    movel([0.504361, -1.310843, -2.623001, -0.778545, 1.570796, 2.075158],accel_mss,speed_ms,0,blend_radius_m)
    movel([0.505882, -1.309678, -2.623708, -0.779003, 1.570796, 2.076678],accel_mss,speed_ms,0,blend_radius_m)
    movel([0.507291, -1.308414, -2.624472, -0.779502, 1.570796, 2.078088],accel_mss,speed_ms,0,blend_radius_m)
    movel([0.508613, -1.307071, -2.625283, -0.780035, 1.570796, 2.079409],accel_mss,speed_ms,0,blend_radius_m)
    movel([0.509871, -1.305667, -2.626128, -0.780594, 1.570796, 2.080667],accel_mss,speed_ms,0,blend_radius_m)
    movel([0.514730, -1.299885, -2.629580, -0.782925, 1.570796, 2.085526],accel_mss,speed_ms,0,blend_radius_m)
    movel([0.516568, -1.297775, -2.630828, -0.783786, 1.570796, 2.087364],accel_mss,speed_ms,0,blend_radius_m)
    movel([0.518895, -1.295391, -2.632232, -0.784766, 1.570796, 2.089692],accel_mss,speed_ms,0,blend_radius_m)
    movel([0.520143, -1.294383, -2.632824, -0.785183, 1.570796, 2.090940],accel_mss,speed_ms,0,blend_radius_m)
    movel([0.521391, -1.293655, -2.633250, -0.785484, 1.570796, 2.092187],accel_mss,speed_ms,0,blend_radius_m)
    movel([0.522003, -1.293434, -2.633379, -0.785576, 1.570796, 2.092800],accel_mss,speed_ms,0,blend_radius_m)
    movel([0.523177, -1.293343, -2.633433, -0.785614, 1.570796, 2.093973],accel_mss,speed_ms,0,blend_radius_m)
    movel([0.523727, -1.293507, -2.633336, -0.785546, 1.570796, 2.094523],accel_mss,speed_ms,0,blend_radius_m)
    movel([0.524119, -1.293909, -2.633101, -0.785379, 1.570796, 2.094915],accel_mss,speed_ms,0,blend_radius_m)
    movel([0.524203, -1.294537, -2.632733, -0.785119, 1.570796, 2.095000],accel_mss,speed_ms,0,blend_radius_m)
    movel([0.523804, -1.296075, -2.631830, -0.784484, 1.570796, 2.094600],accel_mss,speed_ms,0,blend_radius_m)
    movel([0.522876, -1.298205, -2.630574, -0.783610, 1.570796, 2.093672],accel_mss,speed_ms,0,blend_radius_m)
    movel([0.521782, -1.300323, -2.629319, -0.782746, 1.570796, 2.092578],accel_mss,speed_ms,0,blend_radius_m)
    movel([0.523955, -1.298870, -2.630181, -0.783338, 1.570796, 2.094752],accel_mss,speed_ms,0,blend_radius_m)
    movel([0.526201, -1.297582, -2.630942, -0.783865, 1.570796, 2.096997],accel_mss,speed_ms,0,blend_radius_m)
    movel([0.528485, -1.296466, -2.631600, -0.784323, 1.570796, 2.099281],accel_mss,speed_ms,0,blend_radius_m)
    movel([0.530768, -1.295526, -2.632153, -0.784710, 1.570796, 2.101564],accel_mss,speed_ms,0,blend_radius_m)
    movel([0.535321, -1.293655, -2.633250, -0.785484, 1.570796, 2.106117],accel_mss,speed_ms,0,blend_radius_m)
    movel([0.536592, -1.293226, -2.633501, -0.785662, 1.570796, 2.107388],accel_mss,speed_ms,0,blend_radius_m)
    movel([0.537753, -1.292944, -2.633665, -0.785779, 1.570796, 2.108550],accel_mss,speed_ms,0,blend_radius_m)
    movel([0.538730, -1.292873, -2.633707, -0.785809, 1.570796, 2.109526],accel_mss,speed_ms,0,blend_radius_m)
    movel([0.539439, -1.293071, -2.633591, -0.785727, 1.570796, 2.110235],accel_mss,speed_ms,0,blend_radius_m)
    movel([0.539796, -1.293629, -2.633265, -0.785495, 1.570796, 2.110592],accel_mss,speed_ms,0,blend_radius_m)
    movel([0.539763, -1.294477, -2.632768, -0.785143, 1.570796, 2.110560],accel_mss,speed_ms,0,blend_radius_m)
    movel([0.539417, -1.295518, -2.632157, -0.784713, 1.570796, 2.110214],accel_mss,speed_ms,0,blend_radius_m)
    movel([0.538829, -1.296650, -2.631491, -0.784247, 1.570796, 2.109626],accel_mss,speed_ms,0,blend_radius_m)
    movel([0.538074, -1.297775, -2.630828, -0.783786, 1.570796, 2.108870],accel_mss,speed_ms,0,blend_radius_m)
    movel([0.537226, -1.298794, -2.630226, -0.783369, 1.570796, 2.108023],accel_mss,speed_ms,0,blend_radius_m)
    movel([0.536357, -1.299608, -2.629743, -0.783037, 1.570796, 2.107154],accel_mss,speed_ms,0,blend_radius_m)
    movel([0.535539, -1.300121, -2.629439, -0.782829, 1.570796, 2.106335],accel_mss,speed_ms,0,blend_radius_m)
    movel([0.539564, -1.298618, -2.630330, -0.783441, 1.570796, 2.110360],accel_mss,speed_ms,0,blend_radius_m)
    movel([0.541559, -1.298052, -2.630664, -0.783672, 1.570796, 2.112356],accel_mss,speed_ms,0,blend_radius_m)
    movel([0.543523, -1.297629, -2.630915, -0.783846, 1.570796, 2.114320],accel_mss,speed_ms,0,blend_radius_m)
    movel([0.545439, -1.297358, -2.631074, -0.783957, 1.570796, 2.116236],accel_mss,speed_ms,0,blend_radius_m)
    movel([0.547294, -1.297255, -2.631135, -0.783999, 1.570796, 2.118090],accel_mss,speed_ms,0,blend_radius_m)
    movel([0.549070, -1.297333, -2.631089, -0.783967, 1.570796, 2.119867],accel_mss,speed_ms,0,blend_radius_m)
    movel([0.550755, -1.297601, -2.630931, -0.783857, 1.570796, 2.121552],accel_mss,speed_ms,0,blend_radius_m)
    movel([0.551714, -1.298079, -2.630649, -0.783661, 1.570796, 2.122511],accel_mss,speed_ms,0,blend_radius_m)
    movel([0.552495, -1.298983, -2.630114, -0.783292, 1.570796, 2.123291],accel_mss,speed_ms,0,blend_radius_m)
    movel([0.552726, -1.299550, -2.629778, -0.783061, 1.570796, 2.123522],accel_mss,speed_ms,0,blend_radius_m)
    movel([0.552803, -1.300169, -2.629411, -0.782809, 1.570796, 2.123599],accel_mss,speed_ms,0,blend_radius_m)
    movel([0.552691, -1.300824, -2.629021, -0.782543, 1.570796, 2.123487],accel_mss,speed_ms,0,blend_radius_m)
    movel([0.552350, -1.301497, -2.628621, -0.782270, 1.570796, 2.123146],accel_mss,speed_ms,0,blend_radius_m)
    movel([0.551814, -1.302079, -2.628275, -0.782035, 1.570796, 2.122610],accel_mss,speed_ms,0,blend_radius_m)
    movel([0.551157, -1.302554, -2.627992, -0.781844, 1.570796, 2.121954],accel_mss,speed_ms,0,blend_radius_m)
    movel([0.549592, -1.303332, -2.627527, -0.781530, 1.570796, 2.120389],accel_mss,speed_ms,0,blend_radius_m)
    movel([0.548029, -1.303757, -2.627273, -0.781359, 1.570796, 2.118825],accel_mss,speed_ms,0,blend_radius_m)
    movel([0.546506, -1.303910, -2.627181, -0.781298, 1.570796, 2.117302],accel_mss,speed_ms,0,blend_radius_m)
    movel([0.545064, -1.303868, -2.627206, -0.781315, 1.570796, 2.115860],accel_mss,speed_ms,0,blend_radius_m)
    movel([0.546236, -1.305031, -2.626509, -0.780848, 1.570796, 2.117032],accel_mss,speed_ms,0,blend_radius_m)
    movel([0.547593, -1.306014, -2.625919, -0.780456, 1.570796, 2.118389],accel_mss,speed_ms,0,blend_radius_m)
    movel([0.549117, -1.306810, -2.625440, -0.780139, 1.570796, 2.119913],accel_mss,speed_ms,0,blend_radius_m)
    movel([0.550792, -1.307414, -2.625076, -0.779899, 1.570796, 2.121588],accel_mss,speed_ms,0,blend_radius_m)
    movel([0.552231, -1.307696, -2.624906, -0.779787, 1.570796, 2.123027],accel_mss,speed_ms,0,blend_radius_m)
    movel([0.555218, -1.307960, -2.624746, -0.779682, 1.570796, 2.126015],accel_mss,speed_ms,0,blend_radius_m)
    movel([0.556664, -1.308230, -2.624584, -0.779575, 1.570796, 2.127460],accel_mss,speed_ms,0,blend_radius_m)
    movel([0.558212, -1.308690, -2.624306, -0.779393, 1.570796, 2.129009],accel_mss,speed_ms,0,blend_radius_m)
    movel([0.560696, -1.309649, -2.623725, -0.779015, 1.570796, 2.131492],accel_mss,speed_ms,0,blend_radius_m)
    movel([0.561790, -1.310255, -2.623358, -0.778776, 1.570796, 2.132586],accel_mss,speed_ms,0,blend_radius_m)
    movel([0.562521, -1.310911, -2.622960, -0.778519, 1.570796, 2.133318],accel_mss,speed_ms,0,blend_radius_m)
    movel([0.562691, -1.311249, -2.622754, -0.778386, 1.570796, 2.133487],accel_mss,speed_ms,0,blend_radius_m)
    movel([0.562694, -1.311591, -2.622546, -0.778252, 1.570796, 2.133490],accel_mss,speed_ms,0,blend_radius_m)
    movel([0.562510, -1.311931, -2.622339, -0.778119, 1.570796, 2.133307],accel_mss,speed_ms,0,blend_radius_m)
    movel([0.562113, -1.312265, -2.622135, -0.777989, 1.570796, 2.132910],accel_mss,speed_ms,0,blend_radius_m)
    movel([0.561025, -1.312830, -2.621791, -0.777768, 1.570796, 2.131822],accel_mss,speed_ms,0,blend_radius_m)
    movel([0.559815, -1.313224, -2.621550, -0.777614, 1.570796, 2.130611],accel_mss,speed_ms,0,blend_radius_m)
    movel([0.558524, -1.313482, -2.621393, -0.777514, 1.570796, 2.129320],accel_mss,speed_ms,0,blend_radius_m)
    movel([0.557205, -1.313629, -2.621303, -0.777457, 1.570796, 2.128001],accel_mss,speed_ms,0,blend_radius_m)
    movel([0.554665, -1.313702, -2.621258, -0.777429, 1.570796, 2.125461],accel_mss,speed_ms,0,blend_radius_m)
    movel([0.552577, -1.313666, -2.621280, -0.777443, 1.570796, 2.123374],accel_mss,speed_ms,0,blend_radius_m)
    movel([0.553095, -1.314568, -2.620728, -0.777093, 1.570796, 2.123892],accel_mss,speed_ms,0,blend_radius_m)
    movel([0.553726, -1.315378, -2.620232, -0.776779, 1.570796, 2.124522],accel_mss,speed_ms,0,blend_radius_m)
    movel([0.555262, -1.316761, -2.619382, -0.776246, 1.570796, 2.126058],accel_mss,speed_ms,0,blend_radius_m)
    movel([0.557070, -1.317890, -2.618687, -0.775813, 1.570796, 2.127867],accel_mss,speed_ms,0,blend_radius_m)
    movel([0.559036, -1.318840, -2.618100, -0.775449, 1.570796, 2.129832],accel_mss,speed_ms,0,blend_radius_m)
    movel([0.560750, -1.319486, -2.617700, -0.775203, 1.570796, 2.131546],accel_mss,speed_ms,0,blend_radius_m)
    movel([0.566077, -1.321158, -2.616663, -0.774568, 1.570796, 2.136873],accel_mss,speed_ms,0,blend_radius_m)
    movel([0.566925, -1.321690, -2.616333, -0.774366, 1.570796, 2.137721],accel_mss,speed_ms,0,blend_radius_m)
    movel([0.567404, -1.322414, -2.615882, -0.774093, 1.570796, 2.138201],accel_mss,speed_ms,0,blend_radius_m)
    movel([0.567376, -1.322780, -2.615654, -0.773955, 1.570796, 2.138172],accel_mss,speed_ms,0,blend_radius_m)
    movel([0.567099, -1.323110, -2.615448, -0.773831, 1.570796, 2.137895],accel_mss,speed_ms,0,blend_radius_m)
    movel([0.566520, -1.323378, -2.615281, -0.773730, 1.570796, 2.137317],accel_mss,speed_ms,0,blend_radius_m)
    movel([0.565588, -1.323554, -2.615171, -0.773664, 1.570796, 2.136384],accel_mss,speed_ms,0,blend_radius_m)
    movel([0.564160, -1.323615, -2.615133, -0.773641, 1.570796, 2.134956],accel_mss,speed_ms,0,blend_radius_m)
    movel([0.562620, -1.323495, -2.615208, -0.773686, 1.570796, 2.133416],accel_mss,speed_ms,0,blend_radius_m)
    movel([0.561231, -1.323153, -2.615421, -0.773815, 1.570796, 2.132027],accel_mss,speed_ms,0,blend_radius_m)
    movel([0.560674, -1.322887, -2.615587, -0.773915, 1.570796, 2.131470],accel_mss,speed_ms,0,blend_radius_m)
    movel([0.560257, -1.322548, -2.615798, -0.774042, 1.570796, 2.131053],accel_mss,speed_ms,0,blend_radius_m)
    movel([0.561241, -1.324942, -2.614303, -0.773144, 1.570796, 2.132038],accel_mss,speed_ms,0,blend_radius_m)
    movel([0.562524, -1.327120, -2.612935, -0.772333, 1.570796, 2.133321],accel_mss,speed_ms,0,blend_radius_m)
    movel([0.564045, -1.329119, -2.611675, -0.771595, 1.570796, 2.134841],accel_mss,speed_ms,0,blend_radius_m)
    movel([0.565745, -1.330982, -2.610496, -0.770912, 1.570796, 2.136541],accel_mss,speed_ms,0,blend_radius_m)
    movel([0.569451, -1.334431, -2.608299, -0.769659, 1.570796, 2.140247],accel_mss,speed_ms,0,blend_radius_m)
    movel([0.573175, -1.337754, -2.606167, -0.768468, 1.570796, 2.143972],accel_mss,speed_ms,0,blend_radius_m)
    movel([0.573691, -1.338478, -2.605701, -0.768210, 1.570796, 2.144487],accel_mss,speed_ms,0,blend_radius_m)
    movel([0.573735, -1.338932, -2.605408, -0.768049, 1.570796, 2.144531],accel_mss,speed_ms,0,blend_radius_m)
    movel([0.573528, -1.339439, -2.605080, -0.767869, 1.570796, 2.144324],accel_mss,speed_ms,0,blend_radius_m)
    movel([0.573099, -1.339888, -2.604790, -0.767711, 1.570796, 2.143896],accel_mss,speed_ms,0,blend_radius_m)
    movel([0.571722, -1.340678, -2.604279, -0.767432, 1.570796, 2.142518],accel_mss,speed_ms,0,blend_radius_m)
    movel([0.570874, -1.341000, -2.604070, -0.767318, 1.570796, 2.141670],accel_mss,speed_ms,0,blend_radius_m)
    movel([0.569183, -1.341339, -2.603851, -0.767199, 1.570796, 2.139979],accel_mss,speed_ms,0,blend_radius_m)
    movel([0.567539, -1.341325, -2.603860, -0.767204, 1.570796, 2.138335],accel_mss,speed_ms,0,blend_radius_m)
    movel([0.565973, -1.341026, -2.604053, -0.767309, 1.570796, 2.136769],accel_mss,speed_ms,0,blend_radius_m)
    movel([0.564526, -1.340506, -2.604390, -0.767492, 1.570796, 2.135323],accel_mss,speed_ms,0,blend_radius_m)
    movel([0.563234, -1.339833, -2.604826, -0.767730, 1.570796, 2.134030],accel_mss,speed_ms,0,blend_radius_m)
    movel([0.562135, -1.339068, -2.605320, -0.768001, 1.570796, 2.132931],accel_mss,speed_ms,0,blend_radius_m)
    movel([0.561270, -1.338276, -2.605831, -0.768282, 1.570796, 2.132067],accel_mss,speed_ms,0,blend_radius_m)
    movel([0.561003, -1.338714, -2.605548, -0.768126, 1.570796, 2.131799],accel_mss,speed_ms,0,blend_radius_m)
    movel([0.560974, -1.339164, -2.605258, -0.767967, 1.570796, 2.131770],accel_mss,speed_ms,0,blend_radius_m)
    movel([0.561152, -1.340097, -2.604655, -0.767637, 1.570796, 2.131948],accel_mss,speed_ms,0,blend_radius_m)
    movel([0.561472, -1.340950, -2.604103, -0.767336, 1.570796, 2.132269],accel_mss,speed_ms,0,blend_radius_m)
    movel([0.562363, -1.342502, -2.603095, -0.766792, 1.570796, 2.133160],accel_mss,speed_ms,0,blend_radius_m)
    movel([0.564091, -1.345024, -2.601451, -0.765914, 1.570796, 2.134887],accel_mss,speed_ms,0,blend_radius_m)
    movel([0.565937, -1.347426, -2.599877, -0.765086, 1.570796, 2.136734],accel_mss,speed_ms,0,blend_radius_m)
    movel([0.569942, -1.351936, -2.596899, -0.763554, 1.570796, 2.140738],accel_mss,speed_ms,0,blend_radius_m)
    movel([0.571032, -1.353216, -2.596049, -0.763124, 1.570796, 2.141829],accel_mss,speed_ms,0,blend_radius_m)
    movel([0.571656, -1.354143, -2.595432, -0.762814, 1.570796, 2.142452],accel_mss,speed_ms,0,blend_radius_m)
    movel([0.572170, -1.355176, -2.594743, -0.762470, 1.570796, 2.142967],accel_mss,speed_ms,0,blend_radius_m)
    movel([0.572449, -1.356251, -2.594024, -0.762114, 1.570796, 2.143245],accel_mss,speed_ms,0,blend_radius_m)
    movel([0.572374, -1.357299, -2.593321, -0.761768, 1.570796, 2.143170],accel_mss,speed_ms,0,blend_radius_m)
    movel([0.572168, -1.357794, -2.592990, -0.761606, 1.570796, 2.142964],accel_mss,speed_ms,0,blend_radius_m)
    movel([0.571829, -1.358259, -2.592677, -0.761453, 1.570796, 2.142626],accel_mss,speed_ms,0,blend_radius_m)
    movel([0.571338, -1.358686, -2.592390, -0.761313, 1.570796, 2.142135],accel_mss,speed_ms,0,blend_radius_m)
    movel([0.570686, -1.359068, -2.592133, -0.761188, 1.570796, 2.141483],accel_mss,speed_ms,0,blend_radius_m)
    movel([0.569974, -1.359179, -2.592058, -0.761152, 1.570796, 2.140771],accel_mss,speed_ms,0,blend_radius_m)
    movel([0.569174, -1.359018, -2.592167, -0.761205, 1.570796, 2.139971],accel_mss,speed_ms,0,blend_radius_m)
    movel([0.565202, -1.357551, -2.593152, -0.761685, 1.570796, 2.135998],accel_mss,speed_ms,0,blend_radius_m)
    movel([0.563995, -1.356820, -2.593642, -0.761926, 1.570796, 2.134792],accel_mss,speed_ms,0,blend_radius_m)
    movel([0.563549, -1.356378, -2.593939, -0.762072, 1.570796, 2.134345],accel_mss,speed_ms,0,blend_radius_m)
    movel([0.563259, -1.355871, -2.594278, -0.762240, 1.570796, 2.134055],accel_mss,speed_ms,0,blend_radius_m)
    movel([0.563894, -1.359000, -2.592178, -0.761210, 1.570796, 2.134690],accel_mss,speed_ms,0,blend_radius_m)
    movel([0.564930, -1.361895, -2.590224, -0.760271, 1.570796, 2.135727],accel_mss,speed_ms,0,blend_radius_m)
    movel([0.566288, -1.364581, -2.588399, -0.759409, 1.570796, 2.137084],accel_mss,speed_ms,0,blend_radius_m)
    movel([0.567890, -1.367082, -2.586691, -0.758616, 1.570796, 2.138687],accel_mss,speed_ms,0,blend_radius_m)
    movel([0.569508, -1.368812, -2.585505, -0.758073, 1.570796, 2.140304],accel_mss,speed_ms,0,blend_radius_m)
    movel([0.571786, -1.371355, -2.583753, -0.757281, 1.570796, 2.142582],accel_mss,speed_ms,0,blend_radius_m)
    movel([0.572698, -1.372726, -2.582804, -0.756859, 1.570796, 2.143494],accel_mss,speed_ms,0,blend_radius_m)
    movel([0.573213, -1.374054, -2.581883, -0.756452, 1.570796, 2.144009],accel_mss,speed_ms,0,blend_radius_m)
    movel([0.573263, -1.374675, -2.581452, -0.756263, 1.570796, 2.144060],accel_mss,speed_ms,0,blend_radius_m)
    movel([0.573144, -1.375252, -2.581050, -0.756087, 1.570796, 2.143941],accel_mss,speed_ms,0,blend_radius_m)
    movel([0.572832, -1.375778, -2.580683, -0.755928, 1.570796, 2.143628],accel_mss,speed_ms,0,blend_radius_m)
    movel([0.572309, -1.376242, -2.580360, -0.755787, 1.570796, 2.143105],accel_mss,speed_ms,0,blend_radius_m)
    movel([0.571702, -1.376584, -2.580121, -0.755684, 1.570796, 2.142498],accel_mss,speed_ms,0,blend_radius_m)
    movel([0.571079, -1.376828, -2.579951, -0.755610, 1.570796, 2.141875],accel_mss,speed_ms,0,blend_radius_m)
    movel([0.569831, -1.377119, -2.579747, -0.755523, 1.570796, 2.140627],accel_mss,speed_ms,0,blend_radius_m)
    movel([0.568531, -1.377283, -2.579632, -0.755473, 1.570796, 2.139327],accel_mss,speed_ms,0,blend_radius_m)
    movel([0.566060, -1.377286, -2.579631, -0.755473, 1.570796, 2.136857],accel_mss,speed_ms,0,blend_radius_m)
    movel([0.564904, -1.377127, -2.579742, -0.755520, 1.570796, 2.135700],accel_mss,speed_ms,0,blend_radius_m)
    movel([0.566200, -1.378941, -2.578471, -0.754977, 1.570796, 2.136997],accel_mss,speed_ms,0,blend_radius_m)
    movel([0.567641, -1.380619, -2.577292, -0.754478, 1.570796, 2.138437],accel_mss,speed_ms,0,blend_radius_m)
    movel([0.569208, -1.382177, -2.576193, -0.754019, 1.570796, 2.140004],accel_mss,speed_ms,0,blend_radius_m)
    movel([0.570887, -1.383627, -2.575167, -0.753594, 1.570796, 2.141683],accel_mss,speed_ms,0,blend_radius_m)
    movel([0.574515, -1.386268, -2.573291, -0.752829, 1.570796, 2.145311],accel_mss,speed_ms,0,blend_radius_m)
    movel([0.578407, -1.388652, -2.571589, -0.752148, 1.570796, 2.149203],accel_mss,speed_ms,0,blend_radius_m)
    movel([0.579346, -1.389428, -2.571034, -0.751928, 1.570796, 2.150143],accel_mss,speed_ms,0,blend_radius_m)
    movel([0.579550, -1.389960, -2.570652, -0.751777, 1.570796, 2.150347],accel_mss,speed_ms,0,blend_radius_m)
    movel([0.579414, -1.390611, -2.570185, -0.751594, 1.570796, 2.150210],accel_mss,speed_ms,0,blend_radius_m)
    movel([0.579137, -1.391041, -2.569875, -0.751473, 1.570796, 2.149933],accel_mss,speed_ms,0,blend_radius_m)
    movel([0.578763, -1.391416, -2.569605, -0.751367, 1.570796, 2.149560],accel_mss,speed_ms,0,blend_radius_m)
    movel([0.577769, -1.392026, -2.569166, -0.751197, 1.570796, 2.148566],accel_mss,speed_ms,0,blend_radius_m)
    movel([0.576546, -1.392460, -2.568853, -0.751076, 1.570796, 2.147343],accel_mss,speed_ms,0,blend_radius_m)
    movel([0.575200, -1.392746, -2.568647, -0.750996, 1.570796, 2.145996],accel_mss,speed_ms,0,blend_radius_m)
    movel([0.572584, -1.392961, -2.568492, -0.750936, 1.570796, 2.143381],accel_mss,speed_ms,0,blend_radius_m)
    movel([0.570809, -1.392845, -2.568576, -0.750969, 1.570796, 2.141605],accel_mss,speed_ms,0,blend_radius_m)
    movel([0.571535, -1.393443, -2.568143, -0.750802, 1.570796, 2.142331],accel_mss,speed_ms,0,blend_radius_m)
    movel([0.572349, -1.393945, -2.567780, -0.750663, 1.570796, 2.143145],accel_mss,speed_ms,0,blend_radius_m)
    movel([0.574202, -1.394682, -2.567247, -0.750460, 1.570796, 2.144998],accel_mss,speed_ms,0,blend_radius_m)
    movel([0.576313, -1.395072, -2.566965, -0.750353, 1.570796, 2.147110],accel_mss,speed_ms,0,blend_radius_m)
    movel([0.578620, -1.395143, -2.566913, -0.750333, 1.570796, 2.149417],accel_mss,speed_ms,0,blend_radius_m)
    movel([0.581071, -1.394908, -2.567083, -0.750398, 1.570796, 2.151867],accel_mss,speed_ms,0,blend_radius_m)
    movel([0.583605, -1.394395, -2.567455, -0.750539, 1.570796, 2.154401],accel_mss,speed_ms,0,blend_radius_m)
    movel([0.586169, -1.393616, -2.568018, -0.750754, 1.570796, 2.156965],accel_mss,speed_ms,0,blend_radius_m)
    movel([0.588706, -1.392596, -2.568755, -0.751038, 1.570796, 2.159502],accel_mss,speed_ms,0,blend_radius_m)
    movel([0.589829, -1.392133, -2.569089, -0.751167, 1.570796, 2.160625],accel_mss,speed_ms,0,blend_radius_m)
    movel([0.590366, -1.392015, -2.569174, -0.751200, 1.570796, 2.161163],accel_mss,speed_ms,0,blend_radius_m)
    movel([0.590849, -1.392039, -2.569157, -0.751193, 1.570796, 2.161645],accel_mss,speed_ms,0,blend_radius_m)
    movel([0.591241, -1.392269, -2.568991, -0.751129, 1.570796, 2.162037],accel_mss,speed_ms,0,blend_radius_m)
    movel([0.591481, -1.392641, -2.568723, -0.751025, 1.570796, 2.162277],accel_mss,speed_ms,0,blend_radius_m)
    movel([0.591567, -1.393380, -2.568189, -0.750820, 1.570796, 2.162364],accel_mss,speed_ms,0,blend_radius_m)
    movel([0.591345, -1.394278, -2.567539, -0.750571, 1.570796, 2.162141],accel_mss,speed_ms,0,blend_radius_m)
    movel([0.590881, -1.395278, -2.566815, -0.750296, 1.570796, 2.161677],accel_mss,speed_ms,0,blend_radius_m)
    movel([0.590241, -1.396332, -2.566049, -0.750007, 1.570796, 2.161037],accel_mss,speed_ms,0,blend_radius_m)
    movel([0.588704, -1.398382, -2.564556, -0.749451, 1.570796, 2.159500],accel_mss,speed_ms,0,blend_radius_m)
    movel([0.587266, -1.400014, -2.563363, -0.749012, 1.570796, 2.158063],accel_mss,speed_ms,0,blend_radius_m)
    movel([0.589604, -1.398798, -2.564252, -0.749339, 1.570796, 2.160401],accel_mss,speed_ms,0,blend_radius_m)
    movel([0.591861, -1.397382, -2.565285, -0.749722, 1.570796, 2.162657],accel_mss,speed_ms,0,blend_radius_m)
    movel([0.594018, -1.395784, -2.566448, -0.750157, 1.570796, 2.164815],accel_mss,speed_ms,0,blend_radius_m)
    movel([0.596054, -1.394033, -2.567717, -0.750639, 1.570796, 2.166851],accel_mss,speed_ms,0,blend_radius_m)
    movel([0.597944, -1.392152, -2.569076, -0.751162, 1.570796, 2.168740],accel_mss,speed_ms,0,blend_radius_m)
    movel([0.599672, -1.390163, -2.570506, -0.751720, 1.570796, 2.170468],accel_mss,speed_ms,0,blend_radius_m)
    movel([0.601208, -1.388096, -2.571987, -0.752306, 1.570796, 2.172005],accel_mss,speed_ms,0,blend_radius_m)
    movel([0.602535, -1.385972, -2.573502, -0.752915, 1.570796, 2.173331],accel_mss,speed_ms,0,blend_radius_m)
    movel([0.604026, -1.382955, -2.575643, -0.753791, 1.570796, 2.174823],accel_mss,speed_ms,0,blend_radius_m)
    movel([0.604912, -1.381390, -2.576749, -0.754250, 1.570796, 2.175709],accel_mss,speed_ms,0,blend_radius_m)
    movel([0.605419, -1.380685, -2.577246, -0.754459, 1.570796, 2.176215],accel_mss,speed_ms,0,blend_radius_m)
    movel([0.605977, -1.380066, -2.577681, -0.754642, 1.570796, 2.176773],accel_mss,speed_ms,0,blend_radius_m)
    movel([0.606991, -1.379225, -2.578272, -0.754892, 1.570796, 2.177787],accel_mss,speed_ms,0,blend_radius_m)
    movel([0.607714, -1.378895, -2.578504, -0.754991, 1.570796, 2.178510],accel_mss,speed_ms,0,blend_radius_m)
    movel([0.608206, -1.378963, -2.578456, -0.754970, 1.570796, 2.179003],accel_mss,speed_ms,0,blend_radius_m)
    movel([0.608528, -1.379314, -2.578209, -0.754866, 1.570796, 2.179324],accel_mss,speed_ms,0,blend_radius_m)
    movel([0.609045, -1.380931, -2.577072, -0.754386, 1.570796, 2.179841],accel_mss,speed_ms,0,blend_radius_m)
    movel([0.609266, -1.381278, -2.576827, -0.754283, 1.570796, 2.180062],accel_mss,speed_ms,0,blend_radius_m)
    movel([0.610734, -1.380000, -2.577727, -0.754662, 1.570796, 2.181531],accel_mss,speed_ms,0,blend_radius_m)
    movel([0.612120, -1.378620, -2.578696, -0.755073, 1.570796, 2.182916],accel_mss,speed_ms,0,blend_radius_m)
    movel([0.613422, -1.377152, -2.579724, -0.755513, 1.570796, 2.184219],accel_mss,speed_ms,0,blend_radius_m)
    movel([0.614645, -1.375605, -2.580804, -0.755980, 1.570796, 2.185441],accel_mss,speed_ms,0,blend_radius_m)
    movel([0.615782, -1.373995, -2.581924, -0.756470, 1.570796, 2.186578],accel_mss,speed_ms,0,blend_radius_m)
    movel([0.616837, -1.372330, -2.583079, -0.756981, 1.570796, 2.187633],accel_mss,speed_ms,0,blend_radius_m)
    movel([0.618706, -1.368889, -2.585451, -0.758048, 1.570796, 2.189502],accel_mss,speed_ms,0,blend_radius_m)
    movel([0.620245, -1.365388, -2.587849, -0.759152, 1.570796, 2.191041],accel_mss,speed_ms,0,blend_radius_m)
    movel([0.621460, -1.361927, -2.590202, -0.760260, 1.570796, 2.192256],accel_mss,speed_ms,0,blend_radius_m)
    movel([0.622342, -1.358612, -2.592439, -0.761337, 1.570796, 2.193139],accel_mss,speed_ms,0,blend_radius_m)
    movel([0.622897, -1.355551, -2.594492, -0.762346, 1.570796, 2.193694],accel_mss,speed_ms,0,blend_radius_m)
    speed_ms = 0.005
    movel([0.622897, -1.346560, -2.590392, -0.775437, 1.570796, 2.193694],accel_mss,speed_ms,0,blend_radius_m)
    speed_ms = 0.040
    movel([0.610502, -1.345377, -2.591171, -0.775841, 1.570796, 2.181298],accel_mss,speed_ms,0,blend_radius_m)
    speed_ms = 0.005
    movel([0.610502, -1.354376, -2.595276, -0.762737, 1.570796, 2.181298],accel_mss,speed_ms,0,blend_radius_m)
    speed_ms = 0.025
    movel([0.610066, -1.353065, -2.596149, -0.763175, 1.570796, 2.180862],accel_mss,speed_ms,0,blend_radius_m)
    movel([0.609319, -1.351998, -2.596858, -0.763533, 1.570796, 2.180115],accel_mss,speed_ms,0,blend_radius_m)
    movel([0.608310, -1.351150, -2.597420, -0.763819, 1.570796, 2.179106],accel_mss,speed_ms,0,blend_radius_m)
    movel([0.607093, -1.350494, -2.597854, -0.764041, 1.570796, 2.177889],accel_mss,speed_ms,0,blend_radius_m)
    movel([0.605719, -1.350002, -2.598179, -0.764207, 1.570796, 2.176515],accel_mss,speed_ms,0,blend_radius_m)
    movel([0.604238, -1.349647, -2.598414, -0.764328, 1.570796, 2.175034],accel_mss,speed_ms,0,blend_radius_m)
    movel([0.601170, -1.349236, -2.598685, -0.764468, 1.570796, 2.171966],accel_mss,speed_ms,0,blend_radius_m)
    speed_ms = 0.005
    movel([0.601170, -1.340202, -2.594557, -0.777630, 1.570796, 2.171966],accel_mss,speed_ms,0,blend_radius_m)
    speed_ms = 0.040
    movel([0.605361, -1.340299, -2.594494, -0.777596, 1.570796, 2.176157],accel_mss,speed_ms,0,blend_radius_m)
    speed_ms = 0.005
    movel([0.605361, -1.349332, -2.598622, -0.764435, 1.570796, 2.176157],accel_mss,speed_ms,0,blend_radius_m)
    speed_ms = 0.025
    movel([0.606903, -1.347649, -2.599730, -0.765010, 1.570796, 2.177699],accel_mss,speed_ms,0,blend_radius_m)
    movel([0.608271, -1.345949, -2.600846, -0.765595, 1.570796, 2.179067],accel_mss,speed_ms,0,blend_radius_m)
    movel([0.609470, -1.344228, -2.601971, -0.766190, 1.570796, 2.180267],accel_mss,speed_ms,0,blend_radius_m)
    movel([0.610511, -1.342486, -2.603105, -0.766797, 1.570796, 2.181308],accel_mss,speed_ms,0,blend_radius_m)
    movel([0.611405, -1.340723, -2.604250, -0.767416, 1.570796, 2.182201],accel_mss,speed_ms,0,blend_radius_m)
    movel([0.612159, -1.338937, -2.605405, -0.768047, 1.570796, 2.182955],accel_mss,speed_ms,0,blend_radius_m)
    movel([0.612782, -1.337127, -2.606570, -0.768691, 1.570796, 2.183579],accel_mss,speed_ms,0,blend_radius_m)
    movel([0.613285, -1.335293, -2.607747, -0.769349, 1.570796, 2.184082],accel_mss,speed_ms,0,blend_radius_m)
    movel([0.614347, -1.329963, -2.611141, -0.771285, 1.570796, 2.185143],accel_mss,speed_ms,0,blend_radius_m)
    movel([0.614957, -1.327383, -2.612770, -0.772236, 1.570796, 2.185753],accel_mss,speed_ms,0,blend_radius_m)
    movel([0.615950, -1.324518, -2.614568, -0.773302, 1.570796, 2.186746],accel_mss,speed_ms,0,blend_radius_m)
    movel([0.617539, -1.320905, -2.616820, -0.774663, 1.570796, 2.188336],accel_mss,speed_ms,0,blend_radius_m)
    movel([0.619412, -1.317279, -2.619063, -0.776047, 1.570796, 2.190208],accel_mss,speed_ms,0,blend_radius_m)
    movel([0.621631, -1.313688, -2.621267, -0.777434, 1.570796, 2.192427],accel_mss,speed_ms,0,blend_radius_m)
    movel([0.622890, -1.311921, -2.622345, -0.778123, 1.570796, 2.193686],accel_mss,speed_ms,0,blend_radius_m)
    movel([0.624259, -1.310184, -2.623400, -0.778804, 1.570796, 2.195056],accel_mss,speed_ms,0,blend_radius_m)
    movel([0.626580, -1.307633, -2.624944, -0.779812, 1.570796, 2.197376],accel_mss,speed_ms,0,blend_radius_m)
    movel([0.629067, -1.305352, -2.626317, -0.780720, 1.570796, 2.199863],accel_mss,speed_ms,0,blend_radius_m)
    movel([0.631695, -1.303353, -2.627514, -0.781522, 1.570796, 2.202491],accel_mss,speed_ms,0,blend_radius_m)
    movel([0.634436, -1.301648, -2.628531, -0.782209, 1.570796, 2.205232],accel_mss,speed_ms,0,blend_radius_m)
    movel([0.637256, -1.300253, -2.629361, -0.782775, 1.570796, 2.208052],accel_mss,speed_ms,0,blend_radius_m)
    movel([0.640128, -1.299181, -2.629997, -0.783211, 1.570796, 2.210925],accel_mss,speed_ms,0,blend_radius_m)
    movel([0.643026, -1.298442, -2.630434, -0.783513, 1.570796, 2.213822],accel_mss,speed_ms,0,blend_radius_m)
    movel([0.645914, -1.298048, -2.630667, -0.783674, 1.570796, 2.216711],accel_mss,speed_ms,0,blend_radius_m)
    movel([0.648024, -1.297993, -2.630700, -0.783697, 1.570796, 2.218820],accel_mss,speed_ms,0,blend_radius_m)
    movel([0.650051, -1.298145, -2.630609, -0.783634, 1.570796, 2.220848],accel_mss,speed_ms,0,blend_radius_m)
    movel([0.651979, -1.298499, -2.630400, -0.783490, 1.570796, 2.222776],accel_mss,speed_ms,0,blend_radius_m)
    movel([0.653801, -1.299040, -2.630080, -0.783269, 1.570796, 2.224597],accel_mss,speed_ms,0,blend_radius_m)
    movel([0.655496, -1.299767, -2.629649, -0.782973, 1.570796, 2.226292],accel_mss,speed_ms,0,blend_radius_m)
    movel([0.657053, -1.300666, -2.629116, -0.782607, 1.570796, 2.227849],accel_mss,speed_ms,0,blend_radius_m)
    movel([0.658458, -1.301728, -2.628484, -0.782177, 1.570796, 2.229254],accel_mss,speed_ms,0,blend_radius_m)
    movel([0.659698, -1.302944, -2.627759, -0.781686, 1.570796, 2.230494],accel_mss,speed_ms,0,blend_radius_m)
    movel([0.660758, -1.304304, -2.626945, -0.781140, 1.570796, 2.231554],accel_mss,speed_ms,0,blend_radius_m)
    movel([0.661630, -1.305798, -2.626049, -0.780542, 1.570796, 2.232426],accel_mss,speed_ms,0,blend_radius_m)
    movel([0.662298, -1.307417, -2.625075, -0.779898, 1.570796, 2.233095],accel_mss,speed_ms,0,blend_radius_m)
    movel([0.662753, -1.309151, -2.624027, -0.779211, 1.570796, 2.233549],accel_mss,speed_ms,0,blend_radius_m)
    movel([0.662982, -1.310989, -2.622912, -0.778488, 1.570796, 2.233779],accel_mss,speed_ms,0,blend_radius_m)
    movel([0.662971, -1.312923, -2.621734, -0.777732, 1.570796, 2.233767],accel_mss,speed_ms,0,blend_radius_m)
    movel([0.662713, -1.314939, -2.620501, -0.776949, 1.570796, 2.233509],accel_mss,speed_ms,0,blend_radius_m)
    movel([0.662194, -1.317034, -2.619214, -0.776141, 1.570796, 2.232990],accel_mss,speed_ms,0,blend_radius_m)
    movel([0.661222, -1.319798, -2.617507, -0.775084, 1.570796, 2.232018],accel_mss,speed_ms,0,blend_radius_m)
    movel([0.660038, -1.322566, -2.615787, -0.774036, 1.570796, 2.230834],accel_mss,speed_ms,0,blend_radius_m)
    movel([0.658688, -1.325329, -2.614061, -0.773000, 1.570796, 2.229485],accel_mss,speed_ms,0,blend_radius_m)
    movel([0.657229, -1.328072, -2.612336, -0.771981, 1.570796, 2.228025],accel_mss,speed_ms,0,blend_radius_m)
    movel([0.653850, -1.333959, -2.608600, -0.769830, 1.570796, 2.224647],accel_mss,speed_ms,0,blend_radius_m)
    movel([0.650268, -1.339770, -2.604866, -0.767752, 1.570796, 2.221064],accel_mss,speed_ms,0,blend_radius_m)
    movel([0.646532, -1.345512, -2.601132, -0.765745, 1.570796, 2.217329],accel_mss,speed_ms,0,blend_radius_m)
    movel([0.642701, -1.351180, -2.597400, -0.763809, 1.570796, 2.213498],accel_mss,speed_ms,0,blend_radius_m)
    movel([0.627487, -1.373203, -2.582474, -0.756712, 1.570796, 2.198284],accel_mss,speed_ms,0,blend_radius_m)
    movel([0.620438, -1.383934, -2.574950, -0.753505, 1.570796, 2.191235],accel_mss,speed_ms,0,blend_radius_m)
    movel([0.617107, -1.389270, -2.571147, -0.751972, 1.570796, 2.187903],accel_mss,speed_ms,0,blend_radius_m)
    movel([0.613962, -1.394580, -2.567321, -0.750488, 1.570796, 2.184759],accel_mss,speed_ms,0,blend_radius_m)
    movel([0.611040, -1.399864, -2.563473, -0.749052, 1.570796, 2.181837],accel_mss,speed_ms,0,blend_radius_m)
    movel([0.608382, -1.405119, -2.559605, -0.747665, 1.570796, 2.179179],accel_mss,speed_ms,0,blend_radius_m)
    movel([0.606022, -1.410342, -2.555720, -0.746327, 1.570796, 2.176819],accel_mss,speed_ms,0,blend_radius_m)
    movel([0.604002, -1.415533, -2.551818, -0.745037, 1.570796, 2.174798],accel_mss,speed_ms,0,blend_radius_m)
    movel([0.603351, -1.417541, -2.550299, -0.744549, 1.570796, 2.174148],accel_mss,speed_ms,0,blend_radius_m)
    movel([0.602934, -1.419507, -2.548805, -0.744078, 1.570796, 2.173730],accel_mss,speed_ms,0,blend_radius_m)
    movel([0.602913, -1.421316, -2.547425, -0.743648, 1.570796, 2.173709],accel_mss,speed_ms,0,blend_radius_m)
    movel([0.603103, -1.422127, -2.546805, -0.743457, 1.570796, 2.173899],accel_mss,speed_ms,0,blend_radius_m)
    movel([0.603457, -1.422856, -2.546246, -0.743287, 1.570796, 2.174253],accel_mss,speed_ms,0,blend_radius_m)
    speed_ms = 0.005
    movel([0.603457, -1.414356, -2.542440, -0.755592, 1.570796, 2.174253],accel_mss,speed_ms,0,blend_radius_m)
    speed_ms = 0.040
    movel([0.603863, -1.383508, -2.565076, -0.763806, 1.570796, 2.174659],accel_mss,speed_ms,0,blend_radius_m)
    speed_ms = 0.005
    movel([0.603863, -1.392238, -2.569014, -0.751138, 1.570796, 2.174659],accel_mss,speed_ms,0,blend_radius_m)
    speed_ms = 0.025
    movel([0.603127, -1.392685, -2.568691, -0.751013, 1.570796, 2.173924],accel_mss,speed_ms,0,blend_radius_m)
    movel([0.602452, -1.393269, -2.568270, -0.750851, 1.570796, 2.173248],accel_mss,speed_ms,0,blend_radius_m)
    movel([0.601838, -1.393967, -2.567765, -0.750657, 1.570796, 2.172634],accel_mss,speed_ms,0,blend_radius_m)
    movel([0.601271, -1.394766, -2.567186, -0.750437, 1.570796, 2.172067],accel_mss,speed_ms,0,blend_radius_m)
    movel([0.600275, -1.396590, -2.565862, -0.749937, 1.570796, 2.171071],accel_mss,speed_ms,0,blend_radius_m)
    movel([0.599419, -1.398598, -2.564398, -0.749393, 1.570796, 2.170215],accel_mss,speed_ms,0,blend_radius_m)
    movel([0.597252, -1.404343, -2.560179, -0.747867, 1.570796, 2.168049],accel_mss,speed_ms,0,blend_radius_m)
    movel([0.596512, -1.405711, -2.559167, -0.747512, 1.570796, 2.167309],accel_mss,speed_ms,0,blend_radius_m)
    movel([0.596041, -1.406232, -2.558780, -0.747377, 1.570796, 2.166837],accel_mss,speed_ms,0,blend_radius_m)
    movel([0.595523, -1.406503, -2.558579, -0.747307, 1.570796, 2.166319],accel_mss,speed_ms,0,blend_radius_m)
    movel([0.595134, -1.406544, -2.558549, -0.747296, 1.570796, 2.165930],accel_mss,speed_ms,0,blend_radius_m)
    movel([0.594860, -1.406384, -2.558668, -0.747337, 1.570796, 2.165656],accel_mss,speed_ms,0,blend_radius_m)
    movel([0.594686, -1.406051, -2.558915, -0.747423, 1.570796, 2.165483],accel_mss,speed_ms,0,blend_radius_m)
    movel([0.594599, -1.404973, -2.559712, -0.747703, 1.570796, 2.165395],accel_mss,speed_ms,0,blend_radius_m)
    movel([0.594773, -1.403540, -2.560772, -0.748078, 1.570796, 2.165569],accel_mss,speed_ms,0,blend_radius_m)
    movel([0.595504, -1.400500, -2.563007, -0.748882, 1.570796, 2.166300],accel_mss,speed_ms,0,blend_radius_m)
    movel([0.596090, -1.398758, -2.564281, -0.749349, 1.570796, 2.166886],accel_mss,speed_ms,0,blend_radius_m)
    movel([0.594372, -1.400820, -2.562772, -0.748797, 1.570796, 2.165169],accel_mss,speed_ms,0,blend_radius_m)
    movel([0.592915, -1.402977, -2.561186, -0.748226, 1.570796, 2.163712],accel_mss,speed_ms,0,blend_radius_m)
    movel([0.591689, -1.405202, -2.559544, -0.747644, 1.570796, 2.162485],accel_mss,speed_ms,0,blend_radius_m)
    movel([0.590673, -1.407457, -2.557871, -0.747061, 1.570796, 2.161469],accel_mss,speed_ms,0,blend_radius_m)
    movel([0.589835, -1.409717, -2.556187, -0.746485, 1.570796, 2.160631],accel_mss,speed_ms,0,blend_radius_m)
    movel([0.589156, -1.411947, -2.554518, -0.745924, 1.570796, 2.159953],accel_mss,speed_ms,0,blend_radius_m)
    movel([0.588161, -1.416200, -2.551315, -0.744875, 1.570796, 2.158957],accel_mss,speed_ms,0,blend_radius_m)
    movel([0.587799, -1.417025, -2.550690, -0.744674, 1.570796, 2.158595],accel_mss,speed_ms,0,blend_radius_m)
    movel([0.587486, -1.417336, -2.550454, -0.744599, 1.570796, 2.158282],accel_mss,speed_ms,0,blend_radius_m)
    movel([0.587116, -1.417448, -2.550369, -0.744572, 1.570796, 2.157912],accel_mss,speed_ms,0,blend_radius_m)
    movel([0.586787, -1.417282, -2.550495, -0.744612, 1.570796, 2.157583],accel_mss,speed_ms,0,blend_radius_m)
    movel([0.586231, -1.416604, -2.551009, -0.744776, 1.570796, 2.157027],accel_mss,speed_ms,0,blend_radius_m)
    movel([0.585878, -1.415801, -2.551616, -0.744972, 1.570796, 2.156674],accel_mss,speed_ms,0,blend_radius_m)
    movel([0.585699, -1.414896, -2.552299, -0.745193, 1.570796, 2.156495],accel_mss,speed_ms,0,blend_radius_m)
    movel([0.585677, -1.413906, -2.553045, -0.745437, 1.570796, 2.156473],accel_mss,speed_ms,0,blend_radius_m)
    movel([0.586007, -1.411768, -2.554652, -0.745969, 1.570796, 2.156803],accel_mss,speed_ms,0,blend_radius_m)
    movel([0.586683, -1.409559, -2.556305, -0.746525, 1.570796, 2.157480],accel_mss,speed_ms,0,blend_radius_m)
    movel([0.584424, -1.413569, -2.553299, -0.745521, 1.570796, 2.155220],accel_mss,speed_ms,0,blend_radius_m)
    movel([0.583494, -1.415563, -2.551796, -0.745030, 1.570796, 2.154290],accel_mss,speed_ms,0,blend_radius_m)
    movel([0.582805, -1.417562, -2.550283, -0.744544, 1.570796, 2.153601],accel_mss,speed_ms,0,blend_radius_m)
    movel([0.582532, -1.419260, -2.548993, -0.744136, 1.570796, 2.153328],accel_mss,speed_ms,0,blend_radius_m)
    movel([0.582490, -1.422386, -2.546606, -0.743397, 1.570796, 2.153286],accel_mss,speed_ms,0,blend_radius_m)
    movel([0.582207, -1.424030, -2.545345, -0.743014, 1.570796, 2.153004],accel_mss,speed_ms,0,blend_radius_m)
    movel([0.582086, -1.424369, -2.545085, -0.742935, 1.570796, 2.152883],accel_mss,speed_ms,0,blend_radius_m)
    movel([0.581854, -1.424681, -2.544845, -0.742863, 1.570796, 2.152650],accel_mss,speed_ms,0,blend_radius_m)
    movel([0.581493, -1.424854, -2.544712, -0.742823, 1.570796, 2.152289],accel_mss,speed_ms,0,blend_radius_m)
    movel([0.581028, -1.424852, -2.544713, -0.742824, 1.570796, 2.151824],accel_mss,speed_ms,0,blend_radius_m)
    movel([0.579948, -1.424500, -2.544984, -0.742905, 1.570796, 2.150744],accel_mss,speed_ms,0,blend_radius_m)
    movel([0.578329, -1.423569, -2.545699, -0.743121, 1.570796, 2.149126],accel_mss,speed_ms,0,blend_radius_m)
    movel([0.577960, -1.424862, -2.544706, -0.742821, 1.570796, 2.148756],accel_mss,speed_ms,0,blend_radius_m)
    movel([0.577645, -1.426357, -2.543554, -0.742478, 1.570796, 2.148441],accel_mss,speed_ms,0,blend_radius_m)
    movel([0.577453, -1.428005, -2.542280, -0.742104, 1.570796, 2.148249],accel_mss,speed_ms,0,blend_radius_m)
    movel([0.577452, -1.429760, -2.540919, -0.741710, 1.570796, 2.148248],accel_mss,speed_ms,0,blend_radius_m)
    movel([0.578459, -1.432834, -2.538523, -0.741032, 1.570796, 2.149255],accel_mss,speed_ms,0,blend_radius_m)
    movel([0.578981, -1.434604, -2.537138, -0.740648, 1.570796, 2.149777],accel_mss,speed_ms,0,blend_radius_m)
    movel([0.579054, -1.435266, -2.536618, -0.740505, 1.570796, 2.149851],accel_mss,speed_ms,0,blend_radius_m)
    movel([0.578930, -1.435676, -2.536296, -0.740417, 1.570796, 2.149726],accel_mss,speed_ms,0,blend_radius_m)
    movel([0.578610, -1.435930, -2.536097, -0.740363, 1.570796, 2.149406],accel_mss,speed_ms,0,blend_radius_m)
    movel([0.578244, -1.436091, -2.535970, -0.740328, 1.570796, 2.149040],accel_mss,speed_ms,0,blend_radius_m)
    movel([0.577528, -1.436139, -2.535932, -0.740318, 1.570796, 2.148324],accel_mss,speed_ms,0,blend_radius_m)
    movel([0.577053, -1.435949, -2.536081, -0.740359, 1.570796, 2.147850],accel_mss,speed_ms,0,blend_radius_m)
    movel([0.576639, -1.435645, -2.536321, -0.740424, 1.570796, 2.147435],accel_mss,speed_ms,0,blend_radius_m)
    movel([0.575903, -1.434975, -2.536847, -0.740568, 1.570796, 2.146700],accel_mss,speed_ms,0,blend_radius_m)
    movel([0.575457, -1.436740, -2.535459, -0.740190, 1.570796, 2.146253],accel_mss,speed_ms,0,blend_radius_m)
    movel([0.575152, -1.438476, -2.534090, -0.739824, 1.570796, 2.145948],accel_mss,speed_ms,0,blend_radius_m)
    movel([0.574992, -1.440172, -2.532747, -0.739470, 1.570796, 2.145788],accel_mss,speed_ms,0,blend_radius_m)
    movel([0.574969, -1.441823, -2.531436, -0.739130, 1.570796, 2.145765],accel_mss,speed_ms,0,blend_radius_m)
    movel([0.575168, -1.443368, -2.530206, -0.738815, 1.570796, 2.145964],accel_mss,speed_ms,0,blend_radius_m)
    movel([0.575609, -1.444795, -2.529066, -0.738528, 1.570796, 2.146405],accel_mss,speed_ms,0,blend_radius_m)
    movel([0.576832, -1.447452, -2.526935, -0.738002, 1.570796, 2.147628],accel_mss,speed_ms,0,blend_radius_m)
    movel([0.577055, -1.448296, -2.526256, -0.737837, 1.570796, 2.147851],accel_mss,speed_ms,0,blend_radius_m)
    movel([0.576965, -1.448753, -2.525888, -0.737748, 1.570796, 2.147761],accel_mss,speed_ms,0,blend_radius_m)
    movel([0.576654, -1.449187, -2.525538, -0.737664, 1.570796, 2.147450],accel_mss,speed_ms,0,blend_radius_m)
    movel([0.576237, -1.449464, -2.525315, -0.737610, 1.570796, 2.147034],accel_mss,speed_ms,0,blend_radius_m)
    movel([0.575782, -1.449602, -2.525204, -0.737584, 1.570796, 2.146578],accel_mss,speed_ms,0,blend_radius_m)
    movel([0.574884, -1.449595, -2.525209, -0.737585, 1.570796, 2.145680],accel_mss,speed_ms,0,blend_radius_m)
    movel([0.573821, -1.449344, -2.525411, -0.737633, 1.570796, 2.144617],accel_mss,speed_ms,0,blend_radius_m)
    movel([0.572869, -1.448961, -2.525721, -0.737708, 1.570796, 2.143665],accel_mss,speed_ms,0,blend_radius_m)
    movel([0.572013, -1.448465, -2.526120, -0.737804, 1.570796, 2.142809],accel_mss,speed_ms,0,blend_radius_m)
    movel([0.571243, -1.447873, -2.526597, -0.737919, 1.570796, 2.142039],accel_mss,speed_ms,0,blend_radius_m)
    movel([0.571156, -1.449345, -2.525410, -0.737633, 1.570796, 2.141952],accel_mss,speed_ms,0,blend_radius_m)
    movel([0.571249, -1.450744, -2.524280, -0.737365, 1.570796, 2.142045],accel_mss,speed_ms,0,blend_radius_m)
    movel([0.571531, -1.452045, -2.523227, -0.737117, 1.570796, 2.142327],accel_mss,speed_ms,0,blend_radius_m)
    movel([0.572008, -1.453226, -2.522267, -0.736895, 1.570796, 2.142804],accel_mss,speed_ms,0,blend_radius_m)
    movel([0.572690, -1.454268, -2.521420, -0.736701, 1.570796, 2.143486],accel_mss,speed_ms,0,blend_radius_m)
    movel([0.573586, -1.455151, -2.520700, -0.736538, 1.570796, 2.144382],accel_mss,speed_ms,0,blend_radius_m)
    movel([0.574704, -1.455850, -2.520130, -0.736410, 1.570796, 2.145500],accel_mss,speed_ms,0,blend_radius_m)
    movel([0.576054, -1.456348, -2.519722, -0.736318, 1.570796, 2.146850],accel_mss,speed_ms,0,blend_radius_m)
    speed_ms = 0.005
    movel([0.576054, -1.448109, -2.516058, -0.748222, 1.570796, 2.146850],accel_mss,speed_ms,0,blend_radius_m)
    speed_ms = 0.040
    movel([0.585604, -1.442287, -2.520731, -0.749370, 1.570796, 2.156400],accel_mss,speed_ms,0,blend_radius_m)
    speed_ms = 0.005
    movel([0.585604, -1.450572, -2.524420, -0.737398, 1.570796, 2.156400],accel_mss,speed_ms,0,blend_radius_m)
    speed_ms = 0.025
    movel([0.583814, -1.448240, -2.526302, -0.737848, 1.570796, 2.154611],accel_mss,speed_ms,0,blend_radius_m)
    movel([0.583126, -1.447097, -2.527220, -0.738071, 1.570796, 2.153922],accel_mss,speed_ms,0,blend_radius_m)
    movel([0.582592, -1.445916, -2.528168, -0.738305, 1.570796, 2.153389],accel_mss,speed_ms,0,blend_radius_m)
    movel([0.582226, -1.444649, -2.529183, -0.738557, 1.570796, 2.153022],accel_mss,speed_ms,0,blend_radius_m)
    movel([0.582039, -1.443255, -2.530296, -0.738838, 1.570796, 2.152835],accel_mss,speed_ms,0,blend_radius_m)
    movel([0.582043, -1.441690, -2.531542, -0.739157, 1.570796, 2.152839],accel_mss,speed_ms,0,blend_radius_m)
    movel([0.582253, -1.439911, -2.532954, -0.739524, 1.570796, 2.153050],accel_mss,speed_ms,0,blend_radius_m)
    movel([0.583077, -1.436109, -2.535956, -0.740325, 1.570796, 2.153873],accel_mss,speed_ms,0,blend_radius_m)
    movel([0.584263, -1.432233, -2.538993, -0.741163, 1.570796, 2.155059],accel_mss,speed_ms,0,blend_radius_m)
    movel([0.585769, -1.428306, -2.542047, -0.742036, 1.570796, 2.156566],accel_mss,speed_ms,0,blend_radius_m)
    movel([0.587548, -1.424355, -2.545096, -0.742938, 1.570796, 2.158344],accel_mss,speed_ms,0,blend_radius_m)
    movel([0.589196, -1.421115, -2.547579, -0.743696, 1.570796, 2.159993],accel_mss,speed_ms,0,blend_radius_m)
    movel([0.590996, -1.417874, -2.550046, -0.744469, 1.570796, 2.161792],accel_mss,speed_ms,0,blend_radius_m)
    movel([0.594940, -1.411377, -2.554946, -0.746067, 1.570796, 2.165736],accel_mss,speed_ms,0,blend_radius_m)
    movel([0.609438, -1.388730, -2.571533, -0.752125, 1.570796, 2.180234],accel_mss,speed_ms,0,blend_radius_m)
    movel([0.612520, -1.383868, -2.574997, -0.753524, 1.570796, 2.183317],accel_mss,speed_ms,0,blend_radius_m)
    movel([0.615548, -1.378943, -2.578470, -0.754976, 1.570796, 2.186344],accel_mss,speed_ms,0,blend_radius_m)
    movel([0.618446, -1.373967, -2.581944, -0.756479, 1.570796, 2.189243],accel_mss,speed_ms,0,blend_radius_m)
    movel([0.621146, -1.368941, -2.585416, -0.758032, 1.570796, 2.191942],accel_mss,speed_ms,0,blend_radius_m)
    movel([0.623574, -1.363874, -2.588880, -0.759635, 1.570796, 2.194371],accel_mss,speed_ms,0,blend_radius_m)
    movel([0.625657, -1.358775, -2.592330, -0.761284, 1.570796, 2.196453],accel_mss,speed_ms,0,blend_radius_m)
    movel([0.626927, -1.355048, -2.594828, -0.762513, 1.570796, 2.197723],accel_mss,speed_ms,0,blend_radius_m)
    movel([0.628014, -1.351222, -2.597372, -0.763795, 1.570796, 2.198811],accel_mss,speed_ms,0,blend_radius_m)
    movel([0.628873, -1.347360, -2.599920, -0.765109, 1.570796, 2.199669],accel_mss,speed_ms,0,blend_radius_m)
    movel([0.629455, -1.343522, -2.602432, -0.766436, 1.570796, 2.200252],accel_mss,speed_ms,0,blend_radius_m)
    movel([0.629717, -1.339772, -2.604866, -0.767752, 1.570796, 2.200513],accel_mss,speed_ms,0,blend_radius_m)
    movel([0.629612, -1.336173, -2.607183, -0.769033, 1.570796, 2.200408],accel_mss,speed_ms,0,blend_radius_m)
    movel([0.629087, -1.332796, -2.609342, -0.770251, 1.570796, 2.199883],accel_mss,speed_ms,0,blend_radius_m)
    movel([0.628098, -1.329712, -2.611300, -0.771377, 1.570796, 2.198895],accel_mss,speed_ms,0,blend_radius_m)
    movel([0.627440, -1.328399, -2.612130, -0.771860, 1.570796, 2.198236],accel_mss,speed_ms,0,blend_radius_m)
    movel([0.626623, -1.327191, -2.612891, -0.772307, 1.570796, 2.197419],accel_mss,speed_ms,0,blend_radius_m)
    movel([0.625646, -1.326111, -2.613570, -0.772708, 1.570796, 2.196443],accel_mss,speed_ms,0,blend_radius_m)
    movel([0.624512, -1.325183, -2.614152, -0.773054, 1.570796, 2.195308],accel_mss,speed_ms,0,blend_radius_m)
    movel([0.623225, -1.324426, -2.614626, -0.773337, 1.570796, 2.194021],accel_mss,speed_ms,0,blend_radius_m)
    movel([0.621781, -1.323866, -2.614976, -0.773547, 1.570796, 2.192578],accel_mss,speed_ms,0,blend_radius_m)
    movel([0.620189, -1.323521, -2.615192, -0.773676, 1.570796, 2.190985],accel_mss,speed_ms,0,blend_radius_m)
    movel([0.618447, -1.323417, -2.615256, -0.773715, 1.570796, 2.189243],accel_mss,speed_ms,0,blend_radius_m)
    speed_ms = 0.005
    movel([0.618447, -1.314215, -2.611012, -0.787163, 1.570796, 2.189243],accel_mss,speed_ms,0,blend_radius_m)
    speed_ms = 0.040
    movel([0.619533, -1.300841, -2.619131, -0.792417, 1.570796, 2.190329],accel_mss,speed_ms,0,blend_radius_m)
    speed_ms = 0.005
    movel([0.619533, -1.310126, -2.623436, -0.778827, 1.570796, 2.190329],accel_mss,speed_ms,0,blend_radius_m)
    speed_ms = 0.025
    movel([0.620109, -1.308679, -2.624312, -0.779398, 1.570796, 2.190905],accel_mss,speed_ms,0,blend_radius_m)
    movel([0.620827, -1.307239, -2.625181, -0.779968, 1.570796, 2.191624],accel_mss,speed_ms,0,blend_radius_m)
    movel([0.622599, -1.304391, -2.626893, -0.781105, 1.570796, 2.193395],accel_mss,speed_ms,0,blend_radius_m)
    movel([0.624684, -1.301583, -2.628570, -0.782236, 1.570796, 2.195480],accel_mss,speed_ms,0,blend_radius_m)
    movel([0.626909, -1.298827, -2.630206, -0.783356, 1.570796, 2.197705],accel_mss,speed_ms,0,blend_radius_m)
    speed_ms = 0.005
    movel([0.626909, -1.289474, -2.625850, -0.797065, 1.570796, 2.197705],accel_mss,speed_ms,0,blend_radius_m)
    speed_ms = 0.040
    movel([0.629236, -1.292240, -2.624231, -0.795919, 1.570796, 2.200032],accel_mss,speed_ms,0,blend_radius_m)
    speed_ms = 0.005
    movel([0.629236, -1.301576, -2.628574, -0.782239, 1.570796, 2.200032],accel_mss,speed_ms,0,blend_radius_m)
    speed_ms = 0.025
    movel([0.629448, -1.300276, -2.629348, -0.782766, 1.570796, 2.200244],accel_mss,speed_ms,0,blend_radius_m)
    movel([0.629802, -1.298978, -2.630117, -0.783294, 1.570796, 2.200598],accel_mss,speed_ms,0,blend_radius_m)
    movel([0.630897, -1.296389, -2.631645, -0.784355, 1.570796, 2.201693],accel_mss,speed_ms,0,blend_radius_m)
    movel([0.632440, -1.293836, -2.633144, -0.785409, 1.570796, 2.203236],accel_mss,speed_ms,0,blend_radius_m)
    movel([0.634351, -1.291335, -2.634604, -0.786450, 1.570796, 2.205148],accel_mss,speed_ms,0,blend_radius_m)
    movel([0.636548, -1.288908, -2.636013, -0.787468, 1.570796, 2.207344],accel_mss,speed_ms,0,blend_radius_m)
    movel([0.638945, -1.286578, -2.637359, -0.788452, 1.570796, 2.209741],accel_mss,speed_ms,0,blend_radius_m)
    movel([0.641458, -1.284365, -2.638630, -0.789393, 1.570796, 2.212255],accel_mss,speed_ms,0,blend_radius_m)
    movel([0.644002, -1.282293, -2.639816, -0.790280, 1.570796, 2.214798],accel_mss,speed_ms,0,blend_radius_m)
    speed_ms = 0.005
    movel([0.644002, -1.272846, -2.635384, -0.804159, 1.570796, 2.214798],accel_mss,speed_ms,0,blend_radius_m)
    speed_ms = 0.040
    movel([0.669072, -1.259735, -2.642660, -0.809994, 1.570796, 2.239868],accel_mss,speed_ms,0,blend_radius_m)
    speed_ms = 0.005
    movel([0.669072, -1.269252, -2.647151, -0.795986, 1.570796, 2.239868],accel_mss,speed_ms,0,blend_radius_m)
    speed_ms = 0.025
    movel([0.666960, -1.269846, -2.646821, -0.795721, 1.570796, 2.237757],accel_mss,speed_ms,0,blend_radius_m)
    movel([0.664756, -1.270617, -2.646393, -0.795379, 1.570796, 2.235552],accel_mss,speed_ms,0,blend_radius_m)
    movel([0.662493, -1.271553, -2.645872, -0.794964, 1.570796, 2.233289],accel_mss,speed_ms,0,blend_radius_m)
    movel([0.660197, -1.272645, -2.645263, -0.794481, 1.570796, 2.230993],accel_mss,speed_ms,0,blend_radius_m)
    movel([0.657902, -1.273885, -2.644570, -0.793935, 1.570796, 2.228698],accel_mss,speed_ms,0,blend_radius_m)
    movel([0.655639, -1.275258, -2.643799, -0.793332, 1.570796, 2.226436],accel_mss,speed_ms,0,blend_radius_m)
    movel([0.653438, -1.276760, -2.642954, -0.792675, 1.570796, 2.224235],accel_mss,speed_ms,0,blend_radius_m)
    movel([0.651329, -1.278380, -2.642039, -0.791970, 1.570796, 2.222125],accel_mss,speed_ms,0,blend_radius_m)
    movel([0.649343, -1.280103, -2.641063, -0.791223, 1.570796, 2.220140],accel_mss,speed_ms,0,blend_radius_m)
    movel([0.647509, -1.281924, -2.640026, -0.790439, 1.570796, 2.218305],accel_mss,speed_ms,0,blend_radius_m)
    movel([0.645855, -1.283830, -2.638937, -0.789622, 1.570796, 2.216652],accel_mss,speed_ms,0,blend_radius_m)
    movel([0.644412, -1.285811, -2.637800, -0.788778, 1.570796, 2.215208],accel_mss,speed_ms,0,blend_radius_m)
    movel([0.643209, -1.287858, -2.636620, -0.787911, 1.570796, 2.214005],accel_mss,speed_ms,0,blend_radius_m)
    movel([0.642274, -1.289961, -2.635403, -0.787025, 1.570796, 2.213070],accel_mss,speed_ms,0,blend_radius_m)
    movel([0.641632, -1.292110, -2.634152, -0.786127, 1.570796, 2.212428],accel_mss,speed_ms,0,blend_radius_m)
    movel([0.641312, -1.294297, -2.632874, -0.785218, 1.570796, 2.212108],accel_mss,speed_ms,0,blend_radius_m)
    speed_ms = 0.005
    movel([0.641312, -1.284918, -2.628497, -0.798974, 1.570796, 2.212108],accel_mss,speed_ms,0,blend_radius_m)
    speed_ms = 0.040
    movel([0.651214, -1.282509, -2.629886, -0.799994, 1.570796, 2.222010],accel_mss,speed_ms,0,blend_radius_m)
    speed_ms = 0.005
    movel([0.651214, -1.291902, -2.634274, -0.786213, 1.570796, 2.222010],accel_mss,speed_ms,0,blend_radius_m)
    speed_ms = 0.025
    movel([0.651897, -1.290182, -2.635274, -0.786933, 1.570796, 2.222693],accel_mss,speed_ms,0,blend_radius_m)
    movel([0.652726, -1.288451, -2.636278, -0.787660, 1.570796, 2.223522],accel_mss,speed_ms,0,blend_radius_m)
    movel([0.653690, -1.286727, -2.637273, -0.788389, 1.570796, 2.224486],accel_mss,speed_ms,0,blend_radius_m)
    movel([0.654782, -1.285021, -2.638254, -0.789114, 1.570796, 2.225579],accel_mss,speed_ms,0,blend_radius_m)
    movel([0.655991, -1.283349, -2.639213, -0.789828, 1.570796, 2.226787],accel_mss,speed_ms,0,blend_radius_m)
    movel([0.657310, -1.281724, -2.640140, -0.790525, 1.570796, 2.228106],accel_mss,speed_ms,0,blend_radius_m)
    movel([0.658732, -1.280158, -2.641031, -0.791200, 1.570796, 2.229528],accel_mss,speed_ms,0,blend_radius_m)
    movel([0.660243, -1.278670, -2.641875, -0.791844, 1.570796, 2.231039],accel_mss,speed_ms,0,blend_radius_m)
    movel([0.661835, -1.277271, -2.642666, -0.792452, 1.570796, 2.232631],accel_mss,speed_ms,0,blend_radius_m)
    movel([0.663502, -1.275977, -2.643395, -0.793017, 1.570796, 2.234299],accel_mss,speed_ms,0,blend_radius_m)
    movel([0.665227, -1.274805, -2.644054, -0.793530, 1.570796, 2.236023],accel_mss,speed_ms,0,blend_radius_m)
    movel([0.667007, -1.273766, -2.644636, -0.793987, 1.570796, 2.237804],accel_mss,speed_ms,0,blend_radius_m)
    movel([0.668830, -1.272877, -2.645133, -0.794378, 1.570796, 2.239626],accel_mss,speed_ms,0,blend_radius_m)
    movel([0.670684, -1.272153, -2.645538, -0.794698, 1.570796, 2.241481],accel_mss,speed_ms,0,blend_radius_m)
    movel([0.672560, -1.271611, -2.645840, -0.794938, 1.570796, 2.243356],accel_mss,speed_ms,0,blend_radius_m)
    movel([0.674444, -1.271261, -2.646035, -0.795093, 1.570796, 2.245241],accel_mss,speed_ms,0,blend_radius_m)
    movel([0.676214, -1.271136, -2.646104, -0.795149, 1.570796, 2.247010],accel_mss,speed_ms,0,blend_radius_m)
    movel([0.677859, -1.271228, -2.646053, -0.795108, 1.570796, 2.248656],accel_mss,speed_ms,0,blend_radius_m)
    movel([0.679377, -1.271521, -2.645890, -0.794978, 1.570796, 2.250174],accel_mss,speed_ms,0,blend_radius_m)
    movel([0.680769, -1.272004, -2.645621, -0.794764, 1.570796, 2.251565],accel_mss,speed_ms,0,blend_radius_m)
    movel([0.682031, -1.272660, -2.645254, -0.794474, 1.570796, 2.252827],accel_mss,speed_ms,0,blend_radius_m)
    movel([0.683157, -1.273479, -2.644797, -0.794113, 1.570796, 2.253954],accel_mss,speed_ms,0,blend_radius_m)
    movel([0.684155, -1.274441, -2.644258, -0.793690, 1.570796, 2.254951],accel_mss,speed_ms,0,blend_radius_m)
    movel([0.685014, -1.275535, -2.643644, -0.793211, 1.570796, 2.255810],accel_mss,speed_ms,0,blend_radius_m)
    movel([0.685737, -1.276745, -2.642962, -0.792681, 1.570796, 2.256533],accel_mss,speed_ms,0,blend_radius_m)
    movel([0.686774, -1.279456, -2.641430, -0.791503, 1.570796, 2.257571],accel_mss,speed_ms,0,blend_radius_m)
    movel([0.687082, -1.280926, -2.640595, -0.790868, 1.570796, 2.257879],accel_mss,speed_ms,0,blend_radius_m)
    movel([0.687283, -1.284028, -2.638824, -0.789537, 1.570796, 2.258079],accel_mss,speed_ms,0,blend_radius_m)
    movel([0.687174, -1.285630, -2.637905, -0.788855, 1.570796, 2.257970],accel_mss,speed_ms,0,blend_radius_m)
    movel([0.686921, -1.287246, -2.636973, -0.788169, 1.570796, 2.257718],accel_mss,speed_ms,0,blend_radius_m)
    speed_ms = 0.005
    movel([0.686921, -1.277827, -2.632564, -0.801997, 1.570796, 2.257718],accel_mss,speed_ms,0,blend_radius_m)
    speed_ms = 0.040
    movel([0.686153, -1.291546, -2.624638, -0.796205, 1.570796, 2.256949],accel_mss,speed_ms,0,blend_radius_m)
    speed_ms = 0.005
    movel([0.686153, -1.300886, -2.628985, -0.782518, 1.570796, 2.256949],accel_mss,speed_ms,0,blend_radius_m)
    speed_ms = 0.025
    movel([0.686563, -1.298464, -2.630421, -0.783504, 1.570796, 2.257359],accel_mss,speed_ms,0,blend_radius_m)
    movel([0.686602, -1.296181, -2.631767, -0.784440, 1.570796, 2.257399],accel_mss,speed_ms,0,blend_radius_m)
    movel([0.686283, -1.294070, -2.633007, -0.785312, 1.570796, 2.257079],accel_mss,speed_ms,0,blend_radius_m)
    movel([0.685611, -1.292156, -2.634126, -0.786108, 1.570796, 2.256407],accel_mss,speed_ms,0,blend_radius_m)
    movel([0.684603, -1.290473, -2.635106, -0.786811, 1.570796, 2.255399],accel_mss,speed_ms,0,blend_radius_m)
    movel([0.683264, -1.289050, -2.635931, -0.787408, 1.570796, 2.254061],accel_mss,speed_ms,0,blend_radius_m)
    movel([0.681611, -1.287921, -2.636584, -0.787884, 1.570796, 2.252407],accel_mss,speed_ms,0,blend_radius_m)
    movel([0.679652, -1.287111, -2.637052, -0.788226, 1.570796, 2.250448],accel_mss,speed_ms,0,blend_radius_m)
    movel([0.677407, -1.286654, -2.637315, -0.788420, 1.570796, 2.248203],accel_mss,speed_ms,0,blend_radius_m)
    movel([0.674916, -1.286573, -2.637362, -0.788454, 1.570796, 2.245712],accel_mss,speed_ms,0,blend_radius_m)
    movel([0.672268, -1.286884, -2.637182, -0.788322, 1.570796, 2.243064],accel_mss,speed_ms,0,blend_radius_m)
    movel([0.669552, -1.287613, -2.636762, -0.788014, 1.570796, 2.240348],accel_mss,speed_ms,0,blend_radius_m)
    movel([0.666852, -1.288777, -2.636089, -0.787523, 1.570796, 2.237648],accel_mss,speed_ms,0,blend_radius_m)
    movel([0.665538, -1.289527, -2.635654, -0.787208, 1.570796, 2.236335],accel_mss,speed_ms,0,blend_radius_m)
    movel([0.664263, -1.290390, -2.635154, -0.786846, 1.570796, 2.235059],accel_mss,speed_ms,0,blend_radius_m)
    movel([0.663035, -1.291369, -2.634584, -0.786436, 1.570796, 2.233831],accel_mss,speed_ms,0,blend_radius_m)
    movel([0.661866, -1.292469, -2.633943, -0.785977, 1.570796, 2.232663],accel_mss,speed_ms,0,blend_radius_m)
    movel([0.660768, -1.293687, -2.633231, -0.785471, 1.570796, 2.231564],accel_mss,speed_ms,0,blend_radius_m)
    movel([0.659756, -1.295024, -2.632448, -0.784917, 1.570796, 2.230552],accel_mss,speed_ms,0,blend_radius_m)
    speed_ms = 0.005
    movel([0.659756, -1.285649, -2.628074, -0.798666, 1.570796, 2.230552],accel_mss,speed_ms,0,blend_radius_m)
    speed_ms = 0.040
    movel([0.667434, -1.296086, -2.621962, -0.794341, 1.570796, 2.238230],accel_mss,speed_ms,0,blend_radius_m)
    speed_ms = 0.005
    movel([0.667434, -1.305400, -2.626288, -0.780701, 1.570796, 2.238230],accel_mss,speed_ms,0,blend_radius_m)
    speed_ms = 0.025
    movel([0.669418, -1.304874, -2.626604, -0.780911, 1.570796, 2.240215],accel_mss,speed_ms,0,blend_radius_m)
    movel([0.671310, -1.304654, -2.626736, -0.781000, 1.570796, 2.242106],accel_mss,speed_ms,0,blend_radius_m)
    movel([0.673092, -1.304715, -2.626699, -0.780975, 1.570796, 2.243888],accel_mss,speed_ms,0,blend_radius_m)
    movel([0.674741, -1.305035, -2.626507, -0.780847, 1.570796, 2.245537],accel_mss,speed_ms,0,blend_radius_m)
    movel([0.676240, -1.305588, -2.626175, -0.780626, 1.570796, 2.247036],accel_mss,speed_ms,0,blend_radius_m)
    movel([0.677570, -1.306343, -2.625722, -0.780325, 1.570796, 2.248366],accel_mss,speed_ms,0,blend_radius_m)
    movel([0.678716, -1.307277, -2.625159, -0.779953, 1.570796, 2.249512],accel_mss,speed_ms,0,blend_radius_m)
    movel([0.679657, -1.308360, -2.624505, -0.779524, 1.570796, 2.250453],accel_mss,speed_ms,0,blend_radius_m)
    movel([0.680469, -1.309890, -2.623579, -0.778920, 1.570796, 2.251265],accel_mss,speed_ms,0,blend_radius_m)
    movel([0.680812, -1.311531, -2.622583, -0.778276, 1.570796, 2.251609],accel_mss,speed_ms,0,blend_radius_m)
    movel([0.680741, -1.313269, -2.621523, -0.777597, 1.570796, 2.251537],accel_mss,speed_ms,0,blend_radius_m)
    movel([0.680298, -1.315090, -2.620408, -0.776890, 1.570796, 2.251095],accel_mss,speed_ms,0,blend_radius_m)
    movel([0.679538, -1.316977, -2.619249, -0.776163, 1.570796, 2.250334],accel_mss,speed_ms,0,blend_radius_m)
    movel([0.678505, -1.318918, -2.618051, -0.775419, 1.570796, 2.249301],accel_mss,speed_ms,0,blend_radius_m)
    movel([0.677248, -1.320898, -2.616825, -0.774666, 1.570796, 2.248044],accel_mss,speed_ms,0,blend_radius_m)
    movel([0.675817, -1.322904, -2.615576, -0.773908, 1.570796, 2.246614],accel_mss,speed_ms,0,blend_radius_m)
    speed_ms = 0.005
    movel([0.675817, -1.313698, -2.611330, -0.787361, 1.570796, 2.246614],accel_mss,speed_ms,0,blend_radius_m)
    speed_ms = 0.040
    movel([0.665940, -1.309142, -2.614119, -0.789128, 1.570796, 2.236737],accel_mss,speed_ms,0,blend_radius_m)
    speed_ms = 0.005
    movel([0.665940, -1.318376, -2.618386, -0.775626, 1.570796, 2.236737],accel_mss,speed_ms,0,blend_radius_m)
    speed_ms = 0.025
    movel([0.667189, -1.319166, -2.617898, -0.775325, 1.570796, 2.237985],accel_mss,speed_ms,0,blend_radius_m)
    movel([0.668210, -1.320110, -2.617314, -0.774965, 1.570796, 2.239007],accel_mss,speed_ms,0,blend_radius_m)
    movel([0.669011, -1.321200, -2.616637, -0.774552, 1.570796, 2.239807],accel_mss,speed_ms,0,blend_radius_m)
    movel([0.669605, -1.322415, -2.615881, -0.774093, 1.570796, 2.240401],accel_mss,speed_ms,0,blend_radius_m)
    movel([0.670000, -1.323744, -2.615052, -0.773593, 1.570796, 2.240796],accel_mss,speed_ms,0,blend_radius_m)
    movel([0.670206, -1.325167, -2.614162, -0.773060, 1.570796, 2.241002],accel_mss,speed_ms,0,blend_radius_m)
    movel([0.670235, -1.326674, -2.613216, -0.772499, 1.570796, 2.241031],accel_mss,speed_ms,0,blend_radius_m)
    movel([0.670092, -1.328248, -2.612225, -0.771916, 1.570796, 2.240888],accel_mss,speed_ms,0,blend_radius_m)
    movel([0.669791, -1.329876, -2.611196, -0.771317, 1.570796, 2.240588],accel_mss,speed_ms,0,blend_radius_m)
    movel([0.669343, -1.331542, -2.610139, -0.770707, 1.570796, 2.240139],accel_mss,speed_ms,0,blend_radius_m)
    movel([0.668753, -1.333234, -2.609063, -0.770092, 1.570796, 2.239550],accel_mss,speed_ms,0,blend_radius_m)
    movel([0.668036, -1.334937, -2.607975, -0.769477, 1.570796, 2.238832],accel_mss,speed_ms,0,blend_radius_m)
    movel([0.667196, -1.336639, -2.606884, -0.768866, 1.570796, 2.237993],accel_mss,speed_ms,0,blend_radius_m)
    movel([0.665195, -1.339980, -2.604731, -0.767678, 1.570796, 2.235992],accel_mss,speed_ms,0,blend_radius_m)
    movel([0.664049, -1.341596, -2.603683, -0.767109, 1.570796, 2.234845],accel_mss,speed_ms,0,blend_radius_m)
    movel([0.664256, -1.341009, -2.604065, -0.767316, 1.570796, 2.235052],accel_mss,speed_ms,0,blend_radius_m)
    speed_ms = 0.005
    movel([0.664256, -1.331920, -2.599899, -0.780569, 1.570796, 2.235052],accel_mss,speed_ms,0,blend_radius_m)
    speed_ms = 0.040
    movel([0.669329, -1.341680, -2.593594, -0.777115, 1.570796, 2.240125],accel_mss,speed_ms,0,blend_radius_m)
    speed_ms = 0.005
    movel([0.669329, -1.350703, -2.597716, -0.763970, 1.570796, 2.240125],accel_mss,speed_ms,0,blend_radius_m)
    speed_ms = 0.025
    movel([0.667012, -1.352255, -2.596687, -0.763446, 1.570796, 2.237809],accel_mss,speed_ms,0,blend_radius_m)
    movel([0.664808, -1.353984, -2.595538, -0.762867, 1.570796, 2.235605],accel_mss,speed_ms,0,blend_radius_m)
    movel([0.662701, -1.355833, -2.594304, -0.762253, 1.570796, 2.233497],accel_mss,speed_ms,0,blend_radius_m)
    movel([0.660671, -1.357746, -2.593022, -0.761621, 1.570796, 2.231468],accel_mss,speed_ms,0,blend_radius_m)
    movel([0.658520, -1.359912, -2.591564, -0.760913, 1.570796, 2.229316],accel_mss,speed_ms,0,blend_radius_m)
    movel([0.657534, -1.361038, -2.590803, -0.760548, 1.570796, 2.228330],accel_mss,speed_ms,0,blend_radius_m)
    movel([0.656649, -1.362205, -2.590013, -0.760171, 1.570796, 2.227445],accel_mss,speed_ms,0,blend_radius_m)
    movel([0.655897, -1.363413, -2.589194, -0.759782, 1.570796, 2.226693],accel_mss,speed_ms,0,blend_radius_m)
    movel([0.655325, -1.364636, -2.588362, -0.759391, 1.570796, 2.226121],accel_mss,speed_ms,0,blend_radius_m)
    movel([0.654988, -1.365827, -2.587550, -0.759013, 1.570796, 2.225784],accel_mss,speed_ms,0,blend_radius_m)
    movel([0.654928, -1.366946, -2.586784, -0.758659, 1.570796, 2.225725],accel_mss,speed_ms,0,blend_radius_m)
    movel([0.655311, -1.368509, -2.585713, -0.758167, 1.570796, 2.226108],accel_mss,speed_ms,0,blend_radius_m)
    movel([0.655496, -1.369287, -2.585178, -0.757924, 1.570796, 2.226293],accel_mss,speed_ms,0,blend_radius_m)
    movel([0.655524, -1.370128, -2.584599, -0.757662, 1.570796, 2.226321],accel_mss,speed_ms,0,blend_radius_m)
    movel([0.655238, -1.371196, -2.583862, -0.757331, 1.570796, 2.226035],accel_mss,speed_ms,0,blend_radius_m)
    movel([0.654635, -1.372378, -2.583045, -0.756966, 1.570796, 2.225432],accel_mss,speed_ms,0,blend_radius_m)
    movel([0.653794, -1.373631, -2.582177, -0.756581, 1.570796, 2.224590],accel_mss,speed_ms,0,blend_radius_m)
    movel([0.652789, -1.374910, -2.581288, -0.756191, 1.570796, 2.223585],accel_mss,speed_ms,0,blend_radius_m)
    movel([0.650587, -1.377373, -2.579570, -0.755446, 1.570796, 2.221383],accel_mss,speed_ms,0,blend_radius_m)
    movel([0.644135, -1.383963, -2.574929, -0.753497, 1.570796, 2.214932],accel_mss,speed_ms,0,blend_radius_m)
    movel([0.639695, -1.388489, -2.571706, -0.752194, 1.570796, 2.210491],accel_mss,speed_ms,0,blend_radius_m)
    movel([0.638417, -1.389930, -2.570673, -0.751785, 1.570796, 2.209214],accel_mss,speed_ms,0,blend_radius_m)
    movel([0.637140, -1.391519, -2.569531, -0.751339, 1.570796, 2.207937],accel_mss,speed_ms,0,blend_radius_m)
    movel([0.634709, -1.395002, -2.567015, -0.750372, 1.570796, 2.205506],accel_mss,speed_ms,0,blend_radius_m)
    movel([0.633617, -1.396832, -2.565686, -0.749871, 1.570796, 2.204414],accel_mss,speed_ms,0,blend_radius_m)
    movel([0.632649, -1.398676, -2.564341, -0.749371, 1.570796, 2.203445],accel_mss,speed_ms,0,blend_radius_m)
    movel([0.631834, -1.400502, -2.563006, -0.748882, 1.570796, 2.202630],accel_mss,speed_ms,0,blend_radius_m)
    movel([0.631200, -1.402278, -2.561701, -0.748410, 1.570796, 2.201996],accel_mss,speed_ms,0,blend_radius_m)
    movel([0.630780, -1.403969, -2.560455, -0.747965, 1.570796, 2.201576],accel_mss,speed_ms,0,blend_radius_m)
    movel([0.630598, -1.405550, -2.559286, -0.747553, 1.570796, 2.201395],accel_mss,speed_ms,0,blend_radius_m)
    movel([0.630689, -1.406985, -2.558221, -0.747182, 1.570796, 2.201485],accel_mss,speed_ms,0,blend_radius_m)
    movel([0.631078, -1.408246, -2.557284, -0.746859, 1.570796, 2.201874],accel_mss,speed_ms,0,blend_radius_m)
    movel([0.631793, -1.409302, -2.556497, -0.746590, 1.570796, 2.202590],accel_mss,speed_ms,0,blend_radius_m)
    movel([0.632867, -1.410123, -2.555884, -0.746382, 1.570796, 2.203663],accel_mss,speed_ms,0,blend_radius_m)
    movel([0.634326, -1.410681, -2.555467, -0.746242, 1.570796, 2.205122],accel_mss,speed_ms,0,blend_radius_m)
    movel([0.636200, -1.410945, -2.555268, -0.746175, 1.570796, 2.206996],accel_mss,speed_ms,0,blend_radius_m)
    movel([0.637786, -1.410925, -2.555284, -0.746180, 1.570796, 2.208582],accel_mss,speed_ms,0,blend_radius_m)
    movel([0.639424, -1.410729, -2.555430, -0.746230, 1.570796, 2.210220],accel_mss,speed_ms,0,blend_radius_m)
    movel([0.641107, -1.410385, -2.555688, -0.746316, 1.570796, 2.211903],accel_mss,speed_ms,0,blend_radius_m)
    movel([0.642824, -1.409921, -2.556034, -0.746433, 1.570796, 2.213620],accel_mss,speed_ms,0,blend_radius_m)
    movel([0.646315, -1.408753, -2.556906, -0.746730, 1.570796, 2.217111],accel_mss,speed_ms,0,blend_radius_m)
    movel([0.649813, -1.407458, -2.557870, -0.747061, 1.570796, 2.220609],accel_mss,speed_ms,0,blend_radius_m)
    movel([0.653331, -1.406258, -2.558761, -0.747370, 1.570796, 2.224127],accel_mss,speed_ms,0,blend_radius_m)
    movel([0.655091, -1.405764, -2.559127, -0.747498, 1.570796, 2.225887],accel_mss,speed_ms,0,blend_radius_m)
    movel([0.656821, -1.405383, -2.559410, -0.747597, 1.570796, 2.227617],accel_mss,speed_ms,0,blend_radius_m)
    movel([0.658499, -1.405139, -2.559590, -0.747660, 1.570796, 2.229295],accel_mss,speed_ms,0,blend_radius_m)
    movel([0.660101, -1.405068, -2.559642, -0.747678, 1.570796, 2.230897],accel_mss,speed_ms,0,blend_radius_m)
    movel([0.661602, -1.405196, -2.559548, -0.747645, 1.570796, 2.232399],accel_mss,speed_ms,0,blend_radius_m)
    movel([0.662981, -1.405554, -2.559283, -0.747552, 1.570796, 2.233778],accel_mss,speed_ms,0,blend_radius_m)
    movel([0.665610, -1.406851, -2.558321, -0.747217, 1.570796, 2.236406],accel_mss,speed_ms,0,blend_radius_m)
    movel([0.666547, -1.407202, -2.558060, -0.747127, 1.570796, 2.237343],accel_mss,speed_ms,0,blend_radius_m)
    movel([0.667629, -1.407372, -2.557934, -0.747083, 1.570796, 2.238425],accel_mss,speed_ms,0,blend_radius_m)
    movel([0.668828, -1.407294, -2.557992, -0.747103, 1.570796, 2.239625],accel_mss,speed_ms,0,blend_radius_m)
    movel([0.670052, -1.406927, -2.558265, -0.747197, 1.570796, 2.240849],accel_mss,speed_ms,0,blend_radius_m)
    movel([0.670647, -1.406620, -2.558492, -0.747276, 1.570796, 2.241444],accel_mss,speed_ms,0,blend_radius_m)
    movel([0.671215, -1.406225, -2.558785, -0.747378, 1.570796, 2.242011],accel_mss,speed_ms,0,blend_radius_m)
    speed_ms = 0.005
    movel([0.671215, -1.397599, -2.554908, -0.759882, 1.570796, 2.242011],accel_mss,speed_ms,0,blend_radius_m)
    speed_ms = 0.040
    movel([0.680691, -1.388985, -2.561158, -0.762246, 1.570796, 2.251487],accel_mss,speed_ms,0,blend_radius_m)
    speed_ms = 0.005
    movel([0.680691, -1.397674, -2.565072, -0.749642, 1.570796, 2.251487],accel_mss,speed_ms,0,blend_radius_m)
    speed_ms = 0.025
    movel([0.680883, -1.398010, -2.564828, -0.749551, 1.570796, 2.251680],accel_mss,speed_ms,0,blend_radius_m)
    movel([0.680674, -1.398511, -2.564462, -0.749416, 1.570796, 2.251470],accel_mss,speed_ms,0,blend_radius_m)
    movel([0.680200, -1.399003, -2.564103, -0.749283, 1.570796, 2.250996],accel_mss,speed_ms,0,blend_radius_m)
    movel([0.679605, -1.399318, -2.563872, -0.749199, 1.570796, 2.250401],accel_mss,speed_ms,0,blend_radius_m)
    movel([0.679026, -1.399397, -2.563814, -0.749177, 1.570796, 2.249822],accel_mss,speed_ms,0,blend_radius_m)
    movel([0.678495, -1.399343, -2.563854, -0.749192, 1.570796, 2.249291],accel_mss,speed_ms,0,blend_radius_m)
    movel([0.677488, -1.399100, -2.564032, -0.749257, 1.570796, 2.248284],accel_mss,speed_ms,0,blend_radius_m)
    movel([0.676711, -1.399024, -2.564088, -0.749278, 1.570796, 2.247507],accel_mss,speed_ms,0,blend_radius_m)
    movel([0.675887, -1.399074, -2.564050, -0.749264, 1.570796, 2.246684],accel_mss,speed_ms,0,blend_radius_m)
    movel([0.674136, -1.399477, -2.563756, -0.749156, 1.570796, 2.244932],accel_mss,speed_ms,0,blend_radius_m)
    movel([0.672313, -1.400165, -2.563253, -0.748972, 1.570796, 2.243109],accel_mss,speed_ms,0,blend_radius_m)
    movel([0.670505, -1.400982, -2.562653, -0.748754, 1.570796, 2.241301],accel_mss,speed_ms,0,blend_radius_m)
    movel([0.670073, -1.401213, -2.562483, -0.748692, 1.570796, 2.240869],accel_mss,speed_ms,0,blend_radius_m)
    movel([0.669730, -1.401530, -2.562251, -0.748608, 1.570796, 2.240527],accel_mss,speed_ms,0,blend_radius_m)
    movel([0.669616, -1.401957, -2.561937, -0.748495, 1.570796, 2.240413],accel_mss,speed_ms,0,blend_radius_m)
    movel([0.669756, -1.402325, -2.561667, -0.748398, 1.570796, 2.240552],accel_mss,speed_ms,0,blend_radius_m)
    movel([0.670265, -1.402999, -2.561170, -0.748220, 1.570796, 2.241062],accel_mss,speed_ms,0,blend_radius_m)
    movel([0.670916, -1.403551, -2.560763, -0.748075, 1.570796, 2.241712],accel_mss,speed_ms,0,blend_radius_m)
    movel([0.671691, -1.403981, -2.560446, -0.747962, 1.570796, 2.242488],accel_mss,speed_ms,0,blend_radius_m)
    movel([0.672577, -1.404280, -2.560225, -0.747884, 1.570796, 2.243373],accel_mss,speed_ms,0,blend_radius_m)
    movel([0.673550, -1.404448, -2.560101, -0.747840, 1.570796, 2.244346],accel_mss,speed_ms,0,blend_radius_m)
    movel([0.674597, -1.404478, -2.560079, -0.747832, 1.570796, 2.245393],accel_mss,speed_ms,0,blend_radius_m)
    movel([0.675697, -1.404367, -2.560161, -0.747861, 1.570796, 2.246493],accel_mss,speed_ms,0,blend_radius_m)
    movel([0.676837, -1.404109, -2.560351, -0.747929, 1.570796, 2.247633],accel_mss,speed_ms,0,blend_radius_m)
    movel([0.676413, -1.404676, -2.559932, -0.747781, 1.570796, 2.247210],accel_mss,speed_ms,0,blend_radius_m)
    movel([0.676247, -1.405267, -2.559495, -0.747627, 1.570796, 2.247043],accel_mss,speed_ms,0,blend_radius_m)
    movel([0.676318, -1.405806, -2.559096, -0.747487, 1.570796, 2.247115],accel_mss,speed_ms,0,blend_radius_m)
    movel([0.676606, -1.406219, -2.558790, -0.747380, 1.570796, 2.247403],accel_mss,speed_ms,0,blend_radius_m)
    movel([0.677062, -1.406468, -2.558605, -0.747316, 1.570796, 2.247858],accel_mss,speed_ms,0,blend_radius_m)
    movel([0.677622, -1.406590, -2.558515, -0.747284, 1.570796, 2.248418],accel_mss,speed_ms,0,blend_radius_m)
    movel([0.678903, -1.406555, -2.558541, -0.747293, 1.570796, 2.249699],accel_mss,speed_ms,0,blend_radius_m)
    movel([0.680637, -1.406212, -2.558795, -0.747382, 1.570796, 2.251433],accel_mss,speed_ms,0,blend_radius_m)
    movel([0.682402, -1.405611, -2.559240, -0.747537, 1.570796, 2.253199],accel_mss,speed_ms,0,blend_radius_m)
    movel([0.684148, -1.404776, -2.559859, -0.747755, 1.570796, 2.254944],accel_mss,speed_ms,0,blend_radius_m)
    movel([0.685822, -1.403724, -2.560635, -0.748029, 1.570796, 2.256618],accel_mss,speed_ms,0,blend_radius_m)
    movel([0.686346, -1.403307, -2.560943, -0.748139, 1.570796, 2.257143],accel_mss,speed_ms,0,blend_radius_m)
    movel([0.686712, -1.402817, -2.561304, -0.748268, 1.570796, 2.257508],accel_mss,speed_ms,0,blend_radius_m)
    movel([0.686787, -1.402398, -2.561612, -0.748378, 1.570796, 2.257584],accel_mss,speed_ms,0,blend_radius_m)
    movel([0.686704, -1.402025, -2.561887, -0.748477, 1.570796, 2.257500],accel_mss,speed_ms,0,blend_radius_m)
    movel([0.686178, -1.400920, -2.562699, -0.748770, 1.570796, 2.256975],accel_mss,speed_ms,0,blend_radius_m)
    movel([0.684967, -1.399025, -2.564086, -0.749277, 1.570796, 2.255763],accel_mss,speed_ms,0,blend_radius_m)
    movel([0.684628, -1.397802, -2.564979, -0.749608, 1.570796, 2.255424],accel_mss,speed_ms,0,blend_radius_m)
    movel([0.686712, -1.396981, -2.565578, -0.749831, 1.570796, 2.257509],accel_mss,speed_ms,0,blend_radius_m)
    movel([0.687737, -1.396754, -2.565743, -0.749893, 1.570796, 2.258533],accel_mss,speed_ms,0,blend_radius_m)
    movel([0.688707, -1.396701, -2.565781, -0.749907, 1.570796, 2.259503],accel_mss,speed_ms,0,blend_radius_m)
    movel([0.689312, -1.396793, -2.565714, -0.749882, 1.570796, 2.260109],accel_mss,speed_ms,0,blend_radius_m)
    movel([0.689888, -1.396995, -2.565567, -0.749827, 1.570796, 2.260685],accel_mss,speed_ms,0,blend_radius_m)
    movel([0.690779, -1.397631, -2.565104, -0.749654, 1.570796, 2.261575],accel_mss,speed_ms,0,blend_radius_m)
    movel([0.691061, -1.398318, -2.564603, -0.749468, 1.570796, 2.261857],accel_mss,speed_ms,0,blend_radius_m)
    movel([0.691028, -1.398733, -2.564300, -0.749356, 1.570796, 2.261825],accel_mss,speed_ms,0,blend_radius_m)
    movel([0.690852, -1.399170, -2.563980, -0.749239, 1.570796, 2.261648],accel_mss,speed_ms,0,blend_radius_m)
    movel([0.690426, -1.399699, -2.563593, -0.749096, 1.570796, 2.261223],accel_mss,speed_ms,0,blend_radius_m)
    movel([0.689862, -1.400133, -2.563276, -0.748980, 1.570796, 2.260658],accel_mss,speed_ms,0,blend_radius_m)
    movel([0.688558, -1.400756, -2.562819, -0.748814, 1.570796, 2.259355],accel_mss,speed_ms,0,blend_radius_m)
    speed_ms = 0.005
    movel([0.688558, -1.392089, -2.558918, -0.761382, 1.570796, 2.259355],accel_mss,speed_ms,0,blend_radius_m)
    speed_ms = 0.040
    movel([0.716496, -1.351915, -2.586842, -0.773633, 1.570796, 2.287292],accel_mss,speed_ms,0,blend_radius_m)
    speed_ms = 0.005
    movel([0.716496, -1.360868, -2.590918, -0.760603, 1.570796, 2.287292],accel_mss,speed_ms,0,blend_radius_m)
    speed_ms = 0.025
    movel([0.717258, -1.360764, -2.590989, -0.760636, 1.570796, 2.288054],accel_mss,speed_ms,0,blend_radius_m)
    movel([0.717956, -1.360800, -2.590965, -0.760625, 1.570796, 2.288752],accel_mss,speed_ms,0,blend_radius_m)
    movel([0.718581, -1.360962, -2.590855, -0.760572, 1.570796, 2.289378],accel_mss,speed_ms,0,blend_radius_m)
    movel([0.719585, -1.361618, -2.590411, -0.760360, 1.570796, 2.290381],accel_mss,speed_ms,0,blend_radius_m)
    movel([0.719948, -1.362084, -2.590096, -0.760210, 1.570796, 2.290744],accel_mss,speed_ms,0,blend_radius_m)
    movel([0.720357, -1.363222, -2.589323, -0.759844, 1.570796, 2.291153],accel_mss,speed_ms,0,blend_radius_m)
    movel([0.720360, -1.364536, -2.588430, -0.759423, 1.570796, 2.291156],accel_mss,speed_ms,0,blend_radius_m)
    movel([0.720047, -1.365943, -2.587470, -0.758976, 1.570796, 2.290843],accel_mss,speed_ms,0,blend_radius_m)
    movel([0.719489, -1.367396, -2.586476, -0.758517, 1.570796, 2.290286],accel_mss,speed_ms,0,blend_radius_m)
    movel([0.718758, -1.368847, -2.585480, -0.758061, 1.570796, 2.289554],accel_mss,speed_ms,0,blend_radius_m)
    movel([0.717424, -1.371005, -2.583994, -0.757390, 1.570796, 2.288221],accel_mss,speed_ms,0,blend_radius_m)
    movel([0.715860, -1.373097, -2.582547, -0.756745, 1.570796, 2.286657],accel_mss,speed_ms,0,blend_radius_m)
    movel([0.714092, -1.375092, -2.581162, -0.756136, 1.570796, 2.284888],accel_mss,speed_ms,0,blend_radius_m)
    movel([0.710270, -1.378698, -2.578642, -0.755049, 1.570796, 2.281067],accel_mss,speed_ms,0,blend_radius_m)
    movel([0.709523, -1.379622, -2.577993, -0.754774, 1.570796, 2.280320],accel_mss,speed_ms,0,blend_radius_m)
    movel([0.709071, -1.380588, -2.577314, -0.754487, 1.570796, 2.279868],accel_mss,speed_ms,0,blend_radius_m)
    movel([0.709002, -1.381412, -2.576733, -0.754244, 1.570796, 2.279798],accel_mss,speed_ms,0,blend_radius_m)
    movel([0.709144, -1.382165, -2.576202, -0.754022, 1.570796, 2.279941],accel_mss,speed_ms,0,blend_radius_m)
    movel([0.709330, -1.382908, -2.575677, -0.753805, 1.570796, 2.280126],accel_mss,speed_ms,0,blend_radius_m)
    movel([0.709385, -1.383698, -2.575117, -0.753574, 1.570796, 2.280182],accel_mss,speed_ms,0,blend_radius_m)
    movel([0.709218, -1.384465, -2.574573, -0.753351, 1.570796, 2.280015],accel_mss,speed_ms,0,blend_radius_m)
    movel([0.708871, -1.385254, -2.574013, -0.753122, 1.570796, 2.279667],accel_mss,speed_ms,0,blend_radius_m)
    movel([0.707876, -1.386827, -2.572893, -0.752669, 1.570796, 2.278672],accel_mss,speed_ms,0,blend_radius_m)
    movel([0.706251, -1.389023, -2.571323, -0.752042, 1.570796, 2.277047],accel_mss,speed_ms,0,blend_radius_m)
    movel([0.704515, -1.391169, -2.569783, -0.751437, 1.570796, 2.275312],accel_mss,speed_ms,0,blend_radius_m)
    movel([0.702673, -1.393253, -2.568281, -0.750855, 1.570796, 2.273470],accel_mss,speed_ms,0,blend_radius_m)
    movel([0.700734, -1.395274, -2.566818, -0.750297, 1.570796, 2.271531],accel_mss,speed_ms,0,blend_radius_m)
    movel([0.698706, -1.397219, -2.565404, -0.749766, 1.570796, 2.269502],accel_mss,speed_ms,0,blend_radius_m)
    movel([0.696598, -1.399086, -2.564042, -0.749261, 1.570796, 2.267395],accel_mss,speed_ms,0,blend_radius_m)
    movel([0.694414, -1.400865, -2.562739, -0.748785, 1.570796, 2.265210],accel_mss,speed_ms,0,blend_radius_m)
    movel([0.692163, -1.402553, -2.561498, -0.748337, 1.570796, 2.262959],accel_mss,speed_ms,0,blend_radius_m)
    movel([0.690695, -1.403546, -2.560767, -0.748076, 1.570796, 2.261491],accel_mss,speed_ms,0,blend_radius_m)
    movel([0.689166, -1.404397, -2.560139, -0.747853, 1.570796, 2.259962],accel_mss,speed_ms,0,blend_radius_m)
    movel([0.687647, -1.404971, -2.559714, -0.747704, 1.570796, 2.258444],accel_mss,speed_ms,0,blend_radius_m)
    movel([0.686916, -1.405108, -2.559613, -0.747668, 1.570796, 2.257712],accel_mss,speed_ms,0,blend_radius_m)
    movel([0.686211, -1.405127, -2.559599, -0.747663, 1.570796, 2.257008],accel_mss,speed_ms,0,blend_radius_m)
    speed_ms = 0.005
    movel([0.686211, -1.396492, -2.555717, -0.760179, 1.570796, 2.257008],accel_mss,speed_ms,0,blend_radius_m)
    speed_ms = 0.040
    movel([0.681592, -1.398702, -2.554100, -0.759587, 1.570796, 2.252389],accel_mss,speed_ms,0,blend_radius_m)
    speed_ms = 0.005
    movel([0.681592, -1.407320, -2.557973, -0.747096, 1.570796, 2.252389],accel_mss,speed_ms,0,blend_radius_m)
    speed_ms = 0.025
    movel([0.681484, -1.407835, -2.557590, -0.746964, 1.570796, 2.252280],accel_mss,speed_ms,0,blend_radius_m)
    movel([0.681136, -1.408357, -2.557201, -0.746831, 1.570796, 2.251933],accel_mss,speed_ms,0,blend_radius_m)
    movel([0.680630, -1.408828, -2.556850, -0.746711, 1.570796, 2.251426],accel_mss,speed_ms,0,blend_radius_m)
    movel([0.680041, -1.409185, -2.556584, -0.746620, 1.570796, 2.250837],accel_mss,speed_ms,0,blend_radius_m)
    movel([0.679332, -1.409393, -2.556429, -0.746567, 1.570796, 2.250129],accel_mss,speed_ms,0,blend_radius_m)
    movel([0.678677, -1.409430, -2.556402, -0.746558, 1.570796, 2.249473],accel_mss,speed_ms,0,blend_radius_m)
    movel([0.678045, -1.409441, -2.556393, -0.746555, 1.570796, 2.248841],accel_mss,speed_ms,0,blend_radius_m)
    movel([0.677412, -1.409578, -2.556291, -0.746520, 1.570796, 2.248209],accel_mss,speed_ms,0,blend_radius_m)
    movel([0.676574, -1.410138, -2.555872, -0.746378, 1.570796, 2.247371],accel_mss,speed_ms,0,blend_radius_m)
    movel([0.676161, -1.410463, -2.555630, -0.746297, 1.570796, 2.246957],accel_mss,speed_ms,0,blend_radius_m)
    movel([0.675669, -1.410734, -2.555427, -0.746228, 1.570796, 2.246466],accel_mss,speed_ms,0,blend_radius_m)
    movel([0.674291, -1.411191, -2.555085, -0.746113, 1.570796, 2.245087],accel_mss,speed_ms,0,blend_radius_m)
    movel([0.672989, -1.411429, -2.554907, -0.746054, 1.570796, 2.243785],accel_mss,speed_ms,0,blend_radius_m)
    movel([0.671745, -1.411471, -2.554875, -0.746043, 1.570796, 2.242541],accel_mss,speed_ms,0,blend_radius_m)
    movel([0.670537, -1.411352, -2.554964, -0.746073, 1.570796, 2.241333],accel_mss,speed_ms,0,blend_radius_m)
    movel([0.671198, -1.411343, -2.554971, -0.746075, 1.570796, 2.241994],accel_mss,speed_ms,0,blend_radius_m)
    movel([0.671802, -1.411437, -2.554900, -0.746052, 1.570796, 2.242598],accel_mss,speed_ms,0,blend_radius_m)
    movel([0.672251, -1.411733, -2.554679, -0.745978, 1.570796, 2.243048],accel_mss,speed_ms,0,blend_radius_m)
    movel([0.672389, -1.412243, -2.554296, -0.745850, 1.570796, 2.243185],accel_mss,speed_ms,0,blend_radius_m)
    movel([0.672121, -1.412850, -2.553840, -0.745699, 1.570796, 2.242917],accel_mss,speed_ms,0,blend_radius_m)
    movel([0.671586, -1.413396, -2.553429, -0.745563, 1.570796, 2.242382],accel_mss,speed_ms,0,blend_radius_m)
    movel([0.670928, -1.413792, -2.553132, -0.745466, 1.570796, 2.241724],accel_mss,speed_ms,0,blend_radius_m)
    movel([0.669125, -1.414418, -2.552660, -0.745311, 1.570796, 2.239921],accel_mss,speed_ms,0,blend_radius_m)
    movel([0.668030, -1.414636, -2.552495, -0.745257, 1.570796, 2.238827],accel_mss,speed_ms,0,blend_radius_m)
    movel([0.666973, -1.414730, -2.552425, -0.745234, 1.570796, 2.237769],accel_mss,speed_ms,0,blend_radius_m)
    movel([0.665965, -1.414695, -2.552451, -0.745243, 1.570796, 2.236761],accel_mss,speed_ms,0,blend_radius_m)
    movel([0.667027, -1.414906, -2.552292, -0.745191, 1.570796, 2.237823],accel_mss,speed_ms,0,blend_radius_m)
    movel([0.668207, -1.414974, -2.552241, -0.745174, 1.570796, 2.239003],accel_mss,speed_ms,0,blend_radius_m)
    movel([0.669347, -1.415067, -2.552171, -0.745152, 1.570796, 2.240143],accel_mss,speed_ms,0,blend_radius_m)
    movel([0.670300, -1.415343, -2.551962, -0.745084, 1.570796, 2.241096],accel_mss,speed_ms,0,blend_radius_m)
    movel([0.670495, -1.415563, -2.551796, -0.745030, 1.570796, 2.241292],accel_mss,speed_ms,0,blend_radius_m)
    movel([0.670387, -1.415809, -2.551610, -0.744970, 1.570796, 2.241183],accel_mss,speed_ms,0,blend_radius_m)
    movel([0.669406, -1.416589, -2.551020, -0.744780, 1.570796, 2.240202],accel_mss,speed_ms,0,blend_radius_m)
    movel([0.668616, -1.417053, -2.550668, -0.744667, 1.570796, 2.239412],accel_mss,speed_ms,0,blend_radius_m)
    movel([0.667800, -1.417424, -2.550387, -0.744578, 1.570796, 2.238597],accel_mss,speed_ms,0,blend_radius_m)
    movel([0.666980, -1.417690, -2.550186, -0.744513, 1.570796, 2.237776],accel_mss,speed_ms,0,blend_radius_m)
    movel([0.667350, -1.417655, -2.550212, -0.744522, 1.570796, 2.238146],accel_mss,speed_ms,0,blend_radius_m)
    movel([0.667708, -1.417732, -2.550154, -0.744503, 1.570796, 2.238504],accel_mss,speed_ms,0,blend_radius_m)
    movel([0.668364, -1.418161, -2.549828, -0.744400, 1.570796, 2.239161],accel_mss,speed_ms,0,blend_radius_m)
    movel([0.668893, -1.418849, -2.549306, -0.744235, 1.570796, 2.239689],accel_mss,speed_ms,0,blend_radius_m)
    movel([0.669242, -1.419671, -2.548679, -0.744038, 1.570796, 2.240039],accel_mss,speed_ms,0,blend_radius_m)
    movel([0.669361, -1.420504, -2.548044, -0.743840, 1.570796, 2.240158],accel_mss,speed_ms,0,blend_radius_m)
    movel([0.669200, -1.421221, -2.547497, -0.743671, 1.570796, 2.239996],accel_mss,speed_ms,0,blend_radius_m)
    movel([0.668998, -1.421497, -2.547287, -0.743606, 1.570796, 2.239794],accel_mss,speed_ms,0,blend_radius_m)
    movel([0.668707, -1.421695, -2.547135, -0.743559, 1.570796, 2.239503],accel_mss,speed_ms,0,blend_radius_m)
    movel([0.668320, -1.421806, -2.547050, -0.743533, 1.570796, 2.239116],accel_mss,speed_ms,0,blend_radius_m)
    movel([0.667830, -1.421808, -2.547049, -0.743532, 1.570796, 2.238627],accel_mss,speed_ms,0,blend_radius_m)
    movel([0.667360, -1.421656, -2.547165, -0.743568, 1.570796, 2.238156],accel_mss,speed_ms,0,blend_radius_m)
    movel([0.665959, -1.420331, -2.548177, -0.743881, 1.570796, 2.236755],accel_mss,speed_ms,0,blend_radius_m)
    movel([0.665389, -1.419864, -2.548533, -0.743992, 1.570796, 2.236185],accel_mss,speed_ms,0,blend_radius_m)
    movel([0.664698, -1.419529, -2.548788, -0.744072, 1.570796, 2.235494],accel_mss,speed_ms,0,blend_radius_m)
    movel([0.663302, -1.419335, -2.548935, -0.744118, 1.570796, 2.234098],accel_mss,speed_ms,0,blend_radius_m)
    movel([0.661839, -1.419247, -2.549002, -0.744139, 1.570796, 2.232635],accel_mss,speed_ms,0,blend_radius_m)
    movel([0.661170, -1.419073, -2.549135, -0.744181, 1.570796, 2.231967],accel_mss,speed_ms,0,blend_radius_m)
    movel([0.660624, -1.418750, -2.549380, -0.744258, 1.570796, 2.231421],accel_mss,speed_ms,0,blend_radius_m)
    movel([0.660291, -1.418274, -2.549742, -0.744373, 1.570796, 2.231087],accel_mss,speed_ms,0,blend_radius_m)
    movel([0.660256, -1.417644, -2.550221, -0.744525, 1.570796, 2.231053],accel_mss,speed_ms,0,blend_radius_m)
    movel([0.661222, -1.417167, -2.550582, -0.744640, 1.570796, 2.232018],accel_mss,speed_ms,0,blend_radius_m)
    movel([0.662202, -1.416795, -2.550864, -0.744730, 1.570796, 2.232998],accel_mss,speed_ms,0,blend_radius_m)
    speed_ms = 0.005
    movel([0.662202, -1.408248, -2.547033, -0.757108, 1.570796, 2.232998],accel_mss,speed_ms,0,blend_radius_m)
    speed_ms = 0.040
    movel([0.664688, -1.417771, -2.539849, -0.754769, 1.570796, 2.235485],accel_mss,speed_ms,0,blend_radius_m)
    speed_ms = 0.005
    movel([0.664688, -1.426245, -2.543640, -0.742504, 1.570796, 2.235485],accel_mss,speed_ms,0,blend_radius_m)
    speed_ms = 0.025
    movel([0.665369, -1.425897, -2.543909, -0.742584, 1.570796, 2.236165],accel_mss,speed_ms,0,blend_radius_m)
    movel([0.666044, -1.425831, -2.543959, -0.742599, 1.570796, 2.236840],accel_mss,speed_ms,0,blend_radius_m)
    movel([0.666624, -1.426009, -2.543822, -0.742558, 1.570796, 2.237420],accel_mss,speed_ms,0,blend_radius_m)
    movel([0.667013, -1.426392, -2.543527, -0.742470, 1.570796, 2.237809],accel_mss,speed_ms,0,blend_radius_m)
    movel([0.667181, -1.426909, -2.543127, -0.742352, 1.570796, 2.237977],accel_mss,speed_ms,0,blend_radius_m)
    movel([0.667197, -1.427498, -2.542672, -0.742219, 1.570796, 2.237994],accel_mss,speed_ms,0,blend_radius_m)
    movel([0.666976, -1.428767, -2.541689, -0.741933, 1.570796, 2.237773],accel_mss,speed_ms,0,blend_radius_m)
    movel([0.667693, -1.428202, -2.542127, -0.742060, 1.570796, 2.238489],accel_mss,speed_ms,0,blend_radius_m)
    movel([0.668275, -1.427528, -2.542649, -0.742212, 1.570796, 2.239072],accel_mss,speed_ms,0,blend_radius_m)
    movel([0.668676, -1.426804, -2.543208, -0.742376, 1.570796, 2.239473],accel_mss,speed_ms,0,blend_radius_m)
    movel([0.668860, -1.426086, -2.543763, -0.742540, 1.570796, 2.239657],accel_mss,speed_ms,0,blend_radius_m)
    movel([0.669018, -1.426552, -2.543403, -0.742434, 1.570796, 2.239814],accel_mss,speed_ms,0,blend_radius_m)
    movel([0.669052, -1.427067, -2.543005, -0.742317, 1.570796, 2.239849],accel_mss,speed_ms,0,blend_radius_m)
    movel([0.668825, -1.428197, -2.542131, -0.742061, 1.570796, 2.239621],accel_mss,speed_ms,0,blend_radius_m)
    movel([0.668329, -1.429399, -2.541199, -0.741791, 1.570796, 2.239126],accel_mss,speed_ms,0,blend_radius_m)
    movel([0.667701, -1.430598, -2.540267, -0.741524, 1.570796, 2.238498],accel_mss,speed_ms,0,blend_radius_m)
    movel([0.666855, -1.431859, -2.539285, -0.741245, 1.570796, 2.237652],accel_mss,speed_ms,0,blend_radius_m)
    movel([0.665898, -1.432984, -2.538406, -0.740999, 1.570796, 2.236695],accel_mss,speed_ms,0,blend_radius_m)
    movel([0.664935, -1.434075, -2.537552, -0.740762, 1.570796, 2.235731],accel_mss,speed_ms,0,blend_radius_m)
    movel([0.664067, -1.435237, -2.536641, -0.740511, 1.570796, 2.234863],accel_mss,speed_ms,0,blend_radius_m)
    movel([0.664043, -1.434226, -2.537434, -0.740729, 1.570796, 2.234840],accel_mss,speed_ms,0,blend_radius_m)
    movel([0.663758, -1.433339, -2.538128, -0.740922, 1.570796, 2.234554],accel_mss,speed_ms,0,blend_radius_m)
    movel([0.663211, -1.432622, -2.538689, -0.741078, 1.570796, 2.234007],accel_mss,speed_ms,0,blend_radius_m)
    movel([0.662396, -1.432118, -2.539083, -0.741188, 1.570796, 2.233192],accel_mss,speed_ms,0,blend_radius_m)
    speed_ms = 0.005
    movel([0.662396, -1.423689, -2.535316, -0.753383, 1.570796, 2.233192],accel_mss,speed_ms,0,blend_radius_m)
    speed_ms = 0.040
    movel([0.661287, -1.428317, -2.531736, -0.752336, 1.570796, 2.232084],accel_mss,speed_ms,0,blend_radius_m)
    speed_ms = 0.005
    movel([0.661287, -1.436710, -2.535482, -0.740196, 1.570796, 2.232084],accel_mss,speed_ms,0,blend_radius_m)
    speed_ms = 0.025
    movel([0.660627, -1.438429, -2.534126, -0.739833, 1.570796, 2.231423],accel_mss,speed_ms,0,blend_radius_m)
    movel([0.660227, -1.440114, -2.532793, -0.739482, 1.570796, 2.231023],accel_mss,speed_ms,0,blend_radius_m)
    movel([0.660219, -1.441654, -2.531571, -0.739164, 1.570796, 2.231015],accel_mss,speed_ms,0,blend_radius_m)
    movel([0.660404, -1.442336, -2.531028, -0.739025, 1.570796, 2.231200],accel_mss,speed_ms,0,blend_radius_m)
    movel([0.660736, -1.442944, -2.530544, -0.738901, 1.570796, 2.231533],accel_mss,speed_ms,0,blend_radius_m)
    movel([0.661424, -1.443605, -2.530016, -0.738767, 1.570796, 2.232220],accel_mss,speed_ms,0,blend_radius_m)
    movel([0.662303, -1.444056, -2.529656, -0.738676, 1.570796, 2.233099],accel_mss,speed_ms,0,blend_radius_m)
    movel([0.663331, -1.444348, -2.529423, -0.738618, 1.570796, 2.234127],accel_mss,speed_ms,0,blend_radius_m)
    movel([0.664463, -1.444529, -2.529278, -0.738581, 1.570796, 2.235259],accel_mss,speed_ms,0,blend_radius_m)
    movel([0.666867, -1.444756, -2.529097, -0.738536, 1.570796, 2.237663],accel_mss,speed_ms,0,blend_radius_m)
    movel([0.669163, -1.445132, -2.528797, -0.738461, 1.570796, 2.239959],accel_mss,speed_ms,0,blend_radius_m)
    movel([0.670320, -1.445571, -2.528445, -0.738373, 1.570796, 2.241116],accel_mss,speed_ms,0,blend_radius_m)
    movel([0.671306, -1.446202, -2.527939, -0.738248, 1.570796, 2.242103],accel_mss,speed_ms,0,blend_radius_m)
    movel([0.672112, -1.447001, -2.527298, -0.738090, 1.570796, 2.242908],accel_mss,speed_ms,0,blend_radius_m)
    movel([0.672723, -1.447947, -2.526537, -0.737905, 1.570796, 2.243519],accel_mss,speed_ms,0,blend_radius_m)
    movel([0.673133, -1.449017, -2.525675, -0.737697, 1.570796, 2.243929],accel_mss,speed_ms,0,blend_radius_m)
    movel([0.673330, -1.450191, -2.524728, -0.737471, 1.570796, 2.244127],accel_mss,speed_ms,0,blend_radius_m)
    movel([0.673304, -1.451443, -2.523714, -0.737231, 1.570796, 2.244100],accel_mss,speed_ms,0,blend_radius_m)
    movel([0.673047, -1.452753, -2.522652, -0.736984, 1.570796, 2.243843],accel_mss,speed_ms,0,blend_radius_m)
    speed_ms = 0.005
    movel([0.673047, -1.444485, -2.518973, -0.748931, 1.570796, 2.243843],accel_mss,speed_ms,0,blend_radius_m)
    speed_ms = 0.040
    movel([0.663920, -1.413806, -2.542857, -0.755727, 1.570796, 2.234716],accel_mss,speed_ms,0,blend_radius_m)
    speed_ms = 0.005
    movel([0.663920, -1.422310, -2.546665, -0.743415, 1.570796, 2.234716],accel_mss,speed_ms,0,blend_radius_m)
    speed_ms = 0.025
    movel([0.664232, -1.422921, -2.546196, -0.743272, 1.570796, 2.235028],accel_mss,speed_ms,0,blend_radius_m)
    movel([0.664331, -1.423633, -2.545650, -0.743106, 1.570796, 2.235127],accel_mss,speed_ms,0,blend_radius_m)
    movel([0.664224, -1.424041, -2.545337, -0.743011, 1.570796, 2.235020],accel_mss,speed_ms,0,blend_radius_m)
    movel([0.663991, -1.424450, -2.545022, -0.742916, 1.570796, 2.234787],accel_mss,speed_ms,0,blend_radius_m)
    movel([0.663653, -1.424811, -2.544745, -0.742833, 1.570796, 2.234450],accel_mss,speed_ms,0,blend_radius_m)
    movel([0.663230, -1.425069, -2.544547, -0.742774, 1.570796, 2.234026],accel_mss,speed_ms,0,blend_radius_m)
    movel([0.662403, -1.425335, -2.544341, -0.742712, 1.570796, 2.233199],accel_mss,speed_ms,0,blend_radius_m)
    movel([0.662023, -1.425608, -2.544131, -0.742650, 1.570796, 2.232820],accel_mss,speed_ms,0,blend_radius_m)
    movel([0.661744, -1.425968, -2.543853, -0.742567, 1.570796, 2.232541],accel_mss,speed_ms,0,blend_radius_m)
    movel([0.661445, -1.426772, -2.543234, -0.742384, 1.570796, 2.232241],accel_mss,speed_ms,0,blend_radius_m)
    movel([0.661342, -1.427671, -2.542538, -0.742180, 1.570796, 2.232138],accel_mss,speed_ms,0,blend_radius_m)
    movel([0.661395, -1.428517, -2.541883, -0.741989, 1.570796, 2.232191],accel_mss,speed_ms,0,blend_radius_m)
    movel([0.661599, -1.429298, -2.541277, -0.741814, 1.570796, 2.232395],accel_mss,speed_ms,0,blend_radius_m)
    movel([0.661952, -1.429992, -2.540738, -0.741659, 1.570796, 2.232748],accel_mss,speed_ms,0,blend_radius_m)
    movel([0.661095, -1.430599, -2.540266, -0.741524, 1.570796, 2.231892],accel_mss,speed_ms,0,blend_radius_m)
    movel([0.660340, -1.431290, -2.539728, -0.741371, 1.570796, 2.231136],accel_mss,speed_ms,0,blend_radius_m)
    movel([0.659675, -1.432049, -2.539137, -0.741204, 1.570796, 2.230471],accel_mss,speed_ms,0,blend_radius_m)
    movel([0.659092, -1.432858, -2.538505, -0.741027, 1.570796, 2.229889],accel_mss,speed_ms,0,blend_radius_m)
    movel([0.658145, -1.434563, -2.537170, -0.740656, 1.570796, 2.228941],accel_mss,speed_ms,0,blend_radius_m)
    movel([0.657439, -1.436280, -2.535821, -0.740288, 1.570796, 2.228235],accel_mss,speed_ms,0,blend_radius_m)
    movel([0.656789, -1.437938, -2.534515, -0.739937, 1.570796, 2.227585],accel_mss,speed_ms,0,blend_radius_m)
    movel([0.656351, -1.438748, -2.533874, -0.739766, 1.570796, 2.227147],accel_mss,speed_ms,0,blend_radius_m)
    movel([0.655772, -1.439524, -2.533261, -0.739604, 1.570796, 2.226568],accel_mss,speed_ms,0,blend_radius_m)
    movel([0.654998, -1.440214, -2.532714, -0.739461, 1.570796, 2.225794],accel_mss,speed_ms,0,blend_radius_m)
    movel([0.654099, -1.440724, -2.532309, -0.739356, 1.570796, 2.224896],accel_mss,speed_ms,0,blend_radius_m)
    movel([0.653206, -1.440962, -2.532120, -0.739306, 1.570796, 2.224002],accel_mss,speed_ms,0,blend_radius_m)
    movel([0.652455, -1.440836, -2.532220, -0.739332, 1.570796, 2.223251],accel_mss,speed_ms,0,blend_radius_m)
    movel([0.652404, -1.441597, -2.531616, -0.739176, 1.570796, 2.223200],accel_mss,speed_ms,0,blend_radius_m)
    movel([0.651952, -1.443186, -2.530350, -0.738852, 1.570796, 2.222748],accel_mss,speed_ms,0,blend_radius_m)
    movel([0.651563, -1.443989, -2.529710, -0.738690, 1.570796, 2.222359],accel_mss,speed_ms,0,blend_radius_m)
    movel([0.650501, -1.445544, -2.528467, -0.738379, 1.570796, 2.221298],accel_mss,speed_ms,0,blend_radius_m)
    movel([0.649842, -1.446269, -2.527885, -0.738235, 1.570796, 2.220639],accel_mss,speed_ms,0,blend_radius_m)
    movel([0.649105, -1.446945, -2.527343, -0.738101, 1.570796, 2.219901],accel_mss,speed_ms,0,blend_radius_m)
    speed_ms = 0.005
    movel([0.649105, -1.438632, -2.523639, -0.750118, 1.570796, 2.219901],accel_mss,speed_ms,0,blend_radius_m)
    speed_ms = 0.040
    movel([0.645760, -1.437267, -2.524720, -0.750402, 1.570796, 2.216557],accel_mss,speed_ms,0,blend_radius_m)
    speed_ms = 0.005
    movel([0.645760, -1.445590, -2.528429, -0.738369, 1.570796, 2.216557],accel_mss,speed_ms,0,blend_radius_m)
    speed_ms = 0.025
    movel([0.643810, -1.453903, -2.521717, -0.736769, 1.570796, 2.214606],accel_mss,speed_ms,0,blend_radius_m)
    movel([0.643464, -1.454925, -2.520884, -0.736580, 1.570796, 2.214260],accel_mss,speed_ms,0,blend_radius_m)
    movel([0.643151, -1.455399, -2.520497, -0.736492, 1.570796, 2.213947],accel_mss,speed_ms,0,blend_radius_m)
    movel([0.642699, -1.455792, -2.520177, -0.736420, 1.570796, 2.213495],accel_mss,speed_ms,0,blend_radius_m)
    movel([0.641540, -1.456395, -2.519684, -0.736310, 1.570796, 2.212337],accel_mss,speed_ms,0,blend_radius_m)
    movel([0.641136, -1.456885, -2.519283, -0.736221, 1.570796, 2.211932],accel_mss,speed_ms,0,blend_radius_m)
    movel([0.640933, -1.457428, -2.518838, -0.736122, 1.570796, 2.211729],accel_mss,speed_ms,0,blend_radius_m)
    movel([0.640880, -1.458294, -2.518128, -0.735967, 1.570796, 2.211677],accel_mss,speed_ms,0,blend_radius_m)
    movel([0.641074, -1.459107, -2.517461, -0.735821, 1.570796, 2.211871],accel_mss,speed_ms,0,blend_radius_m)
    movel([0.641650, -1.460607, -2.516226, -0.735556, 1.570796, 2.212446],accel_mss,speed_ms,0,blend_radius_m)
    movel([0.641815, -1.461695, -2.515328, -0.735366, 1.570796, 2.212611],accel_mss,speed_ms,0,blend_radius_m)
    movel([0.641805, -1.463314, -2.513989, -0.735086, 1.570796, 2.212602],accel_mss,speed_ms,0,blend_radius_m)
    movel([0.641650, -1.464070, -2.513362, -0.734957, 1.570796, 2.212446],accel_mss,speed_ms,0,blend_radius_m)
    movel([0.641354, -1.464657, -2.512875, -0.734857, 1.570796, 2.212150],accel_mss,speed_ms,0,blend_radius_m)
    movel([0.641142, -1.464854, -2.512711, -0.734824, 1.570796, 2.211938],accel_mss,speed_ms,0,blend_radius_m)
    movel([0.640882, -1.464971, -2.512614, -0.734804, 1.570796, 2.211678],accel_mss,speed_ms,0,blend_radius_m)
    movel([0.640198, -1.464916, -2.512660, -0.734813, 1.570796, 2.210994],accel_mss,speed_ms,0,blend_radius_m)
    movel([0.639955, -1.465557, -2.512127, -0.734705, 1.570796, 2.210751],accel_mss,speed_ms,0,blend_radius_m)
    movel([0.639866, -1.466277, -2.511527, -0.734585, 1.570796, 2.210662],accel_mss,speed_ms,0,blend_radius_m)
    movel([0.640029, -1.467820, -2.510240, -0.734329, 1.570796, 2.210825],accel_mss,speed_ms,0,blend_radius_m)
    movel([0.640851, -1.470424, -2.508059, -0.733906, 1.570796, 2.211647],accel_mss,speed_ms,0,blend_radius_m)
    movel([0.641506, -1.471581, -2.507086, -0.733721, 1.570796, 2.212302],accel_mss,speed_ms,0,blend_radius_m)
    movel([0.642329, -1.472704, -2.506141, -0.733544, 1.570796, 2.213125],accel_mss,speed_ms,0,blend_radius_m)
    movel([0.642963, -1.473908, -2.505125, -0.733357, 1.570796, 2.213759],accel_mss,speed_ms,0,blend_radius_m)
    movel([0.643099, -1.474574, -2.504561, -0.733254, 1.570796, 2.213895],accel_mss,speed_ms,0,blend_radius_m)
    movel([0.643056, -1.475303, -2.503944, -0.733142, 1.570796, 2.213852],accel_mss,speed_ms,0,blend_radius_m)
    movel([0.642918, -1.475698, -2.503609, -0.733082, 1.570796, 2.213714],accel_mss,speed_ms,0,blend_radius_m)
    movel([0.642669, -1.476082, -2.503284, -0.733024, 1.570796, 2.213466],accel_mss,speed_ms,0,blend_radius_m)
    movel([0.642340, -1.476371, -2.503039, -0.732980, 1.570796, 2.213136],accel_mss,speed_ms,0,blend_radius_m)
